# B&R Automation Studio project NAELD004C00R10L518F00 (part 48)

##### Act_OpsRun.st
```iecst
(** 2019-04-16 **)
ACTION Act_OpsRun:
	Act_LogStep;

	IF p_bOpsTravLifErrCmdUnclmp THEN //from travLif width chk error
		eMagConv2ClpAct :=	MagConv2ClpActStopClpr;

		IF (p_eMagConv2ClpStatus = Done AND p_eMagConv2ClpStat = MagConv2ClpActStopClpr) THEN

			eMagConv2ClpAct	:= MagConv2ClpActIdle;
			bPneuUnclmpDone := TRUE; //to travlif
		END_IF
	END_IF

	IF eGotoOpsStep <> eOpsStep THEN

		CASE eGotoOpsStep OF
			MagConvLDStepSelClampCtrl:
				IF p_bMagOrientChkSenPrep THEN
					//checking orientation of mag
					IF p_bMagHeightDetEn AND p_bMagHeightDetPrep THEN

						IF p_bMag3OrientationChkSen1 AND p_bMagHeightDetSen3 THEN // Magazine Type Check with height Detection Sensor
							eOpsStep := eGotoOpsStep;
						ELSE
							eMagConv2ClpAct :=	MagConv2ClpActStopClpr;

							IF (p_eMagConv2ClpStatus = Done AND p_eMagConv2ClpStat = MagConv2ClpActStopClpr) THEN

								eMagConv2ClpAct	:= MagConv2ClpActIdle;
								eStatus		:= Error;
								udiStatus	:= 10008;	//'Wrong Magazine Orientation Placed Or Wrong Magazine Loaded'
							END_IF
						END_IF

					ELSE

						IF p_bMag3OrientationChkSen1 AND NOT p_bMagHeightDetSen3 THEN //Without Check Height Detection Sensor
							eOpsStep := eGotoOpsStep;
						ELSE
							eMagConv2ClpAct :=	MagConv2ClpActStopClpr;
							eSelClampCtrl := PneuActExt; //unclmp
							IF (p_eMagConv2ClpStatus = Done AND p_eMagConv2ClpStat = MagConv2ClpActStopClpr) THEN

								eMagConv2ClpAct	:= MagConv2ClpActIdle;
								eStatus		:= Error;
								udiStatus	:= 10008;	//'Wrong Magazine Orientation Placed Or Wrong Magazine Loaded'
							END_IF
						END_IF

					END_IF
				ELSE
					eOpsStep	:= eGotoOpsStep;
				END_IF

			MagConvLDStepMagExitClampCtrl: //For Siemen
				IF p_eNtParamCustomerReq = Siemens AND (eOpsStep <> MagConvLDStepMagExtMESStdByChk )
					AND (p_tyLocalBufferStat.bBffrMty OR p_bDISOTAGVReady)
					AND NOT(iMagMESAcptCond < 0)AND p_bMcParamMesRFIDEn THEN
					eOpsStep := MagConvLDStepMagExtMESStdByChk;
					eGotoOpsStep := MagConvLDStepMagExtMESStdByChk; //exit mes
					//ePrevStepBeforeMESStdBy := MagConvLDStepMagExitClampCtrl;
				ELSE
					bExitDelAutoRcp := TRUE; 									//Clear the rcp and calc pitch
					eOpsStep	:= eGotoOpsStep;
				END_IF

			MagConvLDStepMagExitMnl:
				IF p_bRlsMag AND  p_eNtParamCustomerReq = Siemens AND eOpsStep <> MagConvLDStepMagExtMESStdByChk
					AND eOpsStep <> MagConvLDStepMagEntMESStdByChk AND p_bMcParamMesRFIDEn THEN
					eGotoOpsStep := MagConvLDStepMagExtMESStdByChk; //exit mes
				ELSE
					IF eOpsStep = MagConvLDStepMagExtMESStdByChk THEN
						ePrevStepBeforeMESStdBy := MagConvLDStepMagExitMnl;
					END_IF
					IF p_eNtParamCustomerReq = We_Fabricate  AND p_bMcParamMesRFIDEn THEN
						bExitDelAutoRcp := TRUE;
					END_IF
					eOpsStep	:= eGotoOpsStep;
				END_IF

			ELSE
				eOpsStep	:= eGotoOpsStep;

		END_CASE

	END_IF

	IF eOpsStep = eGotoOpsStep THEN

		IF bPaused = FALSE THEN

			CASE eOpsStep OF

				MagSetupULStepInitPneu:
					sStepTxt	:= 'Initializing Pneumatic';

					p_usiMagConv := 3;
					CASE p_usiMagConv OF
						1:
							p_tyLocalBufferStat ACCESS ADR(p_tyBufferStat1);
							p_bLocalMagEntrySen ACCESS ADR(p_bMagEntrySen1);
							p_bLocalBufferMagPresent ACCESS ADR(p_bBufferMagPresent1);
							p_dtLocalBufferMagPresentTm ACCESS ADR(p_dtBufferMagPresentTm1);
						2:
							p_tyLocalBufferStat ACCESS ADR(p_tyBufferStat2);
							p_bLocalMagEntrySen ACCESS ADR(p_bMagEntrySen2);
							p_bLocalBufferMagPresent ACCESS ADR(p_bBufferMagPresent2);
							p_dtLocalBufferMagPresentTm ACCESS ADR(p_dtBufferMagPresentTm2);
						3:
							p_tyLocalBufferStat ACCESS ADR(p_tyBufferStat3);
							p_bLocalMagEntrySen ACCESS ADR(p_bMagEntrySen3);
							p_bLocalBufferMagPresent ACCESS ADR(p_bBufferMagPresent3);
							p_dtLocalBufferMagPresentTm ACCESS ADR(p_dtBufferMagPresentTm3);
						4:
							p_tyLocalBufferStat ACCESS ADR(p_tyBufferStat4);
							p_bLocalMagEntrySen ACCESS ADR(p_bMagEntrySen4);
							p_bLocalBufferMagPresent ACCESS ADR(p_bBufferMagPresent4);
							p_dtLocalBufferMagPresentTm ACCESS ADR(p_dtBufferMagPresentTm4);
					END_CASE
					IF p_bProjLifTravMnlLoad = FALSE THEN
						eSafetyBarAct	:= PneuActExt;
					ELSE
						eGotoOpsStep := MagConvLDStepMagUSComm;
					END_IF
					IF (p_eSafetyBarStatus = Done AND p_eSafetyBarStat = PneuActExt) THEN
						eSafetyBarAct	:= PneuActIdle;
						eGotoOpsStep	:= MagConvLDStepInitMag;

						bPaused	:= p_bStop OR p_bStep;
					END_IF

				MagConvLDStepInitMag:
					sStepTxt	:= 'Initializing Magazine';
					IF p_bProjLifTravMnlLoad = TRUE THEN
						eGotoOpsStep := MagConvLDStepMagUSComm;
					ELSIF bMagExitedWait THEN
						eGotoOpsStep	:= MagConvLDStepMagExitedWait;
						//eGotoOpsStep	:= MagConvLDStepInitMagEnt;
					ELSIF (ePrevStepBeforeMESStdBy = MagConvLDStepMagExitMnl AND p_bLinkDIMagPresentSen3) OR (p_bHCommModChg AND p_bLinkDIMagPresentSen3)THEN
						eGotoOpsStep	:= MagConvLDStepMagExitMnl;
					ELSIF p_bNtParamAutoRcpPrep AND p_bHermesSvyPrep AND p_bMcParamHermesSvyEn THEN
						bHCommModChgDone := TRUE; //to UI
						eGotoOpsStep	:= MagConvLDStepInitMagConv;
					ELSE
						bHCommModChgDone := TRUE; //to UI
						eGotoOpsStep	:= MagConvLDStepInitSetMagFull;
					END_IF

					bPaused	:= p_bStop OR p_bStep;

				MagConvLDStepInitMagEnt:
					sStepTxt	:= 'Initializing Magazine Conveyor';
					eMagConv2ClpAct	:= MagConv2ClpActInit;
					IF (p_eMagConv2ClpStatus = Done AND p_eMagConv2ClpStat = MagConv2ClpActInit) THEN
						eMagConv2ClpAct	:= MagConv2ClpActIdle;
						IF p_bMagConv2ClpHvMag = FALSE THEN
							eGotoOpsStep	:= MagConvLDStepMagUSComm;
						ELSE
							eGotoOpsStep	:= MagConvLDStepInitMagFixClp;
						END_IF
					END_IF

				MagConvLDStepInitMagFixClp:
					sStepTxt	:= 'Initializing Fixed Clamp';
					eMagConv2ClpAct	:= MagConv2ClpActFixClprClamp;
					IF (p_eMagConv2ClpStatus = Done AND p_eMagConv2ClpStat = MagConv2ClpActFixClprClamp) THEN
						eMagConv2ClpAct	:= MagConv2ClpActIdle;
						IF bMagAutoEx THEN
							eDSSOTAct	:= SOTActRun;
						ELSE
							eDSSOTAct	:= SOTActIdle;
						END_IF

						IF p_bDIMagConvCAB717Sen THEN
							bMagSizeLarge := TRUE;
						ELSE
							bMagSizeLarge := FALSE;
						END_IF
						eGotoOpsStep	:= MagConvLDStepSelClampCtrl;
					END_IF

				MagConvLDStepInitSetMagFull	:
					sStepTxt	:= 'Set Magazine Full';
					IF bSetMagFull AND p_tyBufferStat3.diTtlBrdCap = 1 THEN
						eBufferAct := BufferActSetFull;
						IF p_eBufferStat = BufferActSetFull AND p_eBufferStatus = Done THEN
							bSetMagFull := FALSE;
							eBufferAct := BufferActIdle;
							eGotoOpsStep	:= MagConvLDStepInitMagConv;
						END_IF
					ELSIF bSetMagFull AND p_tyBufferStat3.diTtlBrdCap <> 1 THEN
						bSetMagFull := FALSE;
						eBufferAct := BufferActIdle;
						eGotoOpsStep	:= MagConvLDStepInitMagConv;
					ELSE
						bSetMagFull := FALSE;
						eBufferAct := BufferActIdle;
						eGotoOpsStep	:= MagConvLDStepInitMagConv;
					END_IF
					bPaused	:= p_bStop OR p_bStep;

				MagConvLDStepInitMagConv:
					sStepTxt	:= 'Initializing Magazine Conveyor';

					eMagConv2ClpAct	:= MagConv2ClpActInitStopClp;
					eSelClampCtrl := PneuActExt;

					IF (p_eMagConv2ClpStatus = Done AND p_eMagConv2ClpStat = MagConv2ClpActInitStopClp)
						AND (p_eSelClampCtrlStat = PneuActExt AND p_eSelClampCtrlStatus = Done)
						THEN
						eSelClampCtrl	:= PneuActIdle;
						eMagConv2ClpAct	:= MagConv2ClpActIdle;

						IF p_bMagConv2ClpHvMag = FALSE THEN
							eGotoOpsStep	:= MagConvLDStepMagUSComm;
							bExitDelAutoRcp := TRUE;
							usiAccWO := 0;
							ePrevStepBeforeMESStdBy := MagConvLDStepNA; //finish exit from extMes
						ELSE
						//	eGotoOpsStep		:= MagConvLDStepBffrStatChk;
							eGotoOpsStep		:= MagConvLDStepSelClampCtrl;
						END_IF

						bPaused	:= p_bStop OR p_bStep;

					END_IF

				MagConvLDStepSafetyBarExtCtrl:
					eSafetyBarAct	:= PneuActExt;

					IF(p_eSafetyBarStatus = Done AND p_eSafetyBarStat = PneuActExt)
						THEN
						eSafetyBarAct	:= PneuActIdle;
						eGotoOpsStep	:= MagConvLDStepMagUSComm;
					END_IF

				MagConvLDStepMagUSComm:
					sStepTxt	:= 'Communicating AIV And Ready Transport In Magazine';

					eAGVMagAct	:= AGVMagActEnter;
					IF bMagAutoEx THEN
						eUSSOTAct	:= SOTActRun;
					ELSE
						eUSSOTAct	:= SOTActIdle;
					END_IF
					eDSSOTAct	:= SOTActIdle;
					bMagSizeLarge := FALSE;
					bMagExitedWait	:= FALSE;

					IF p_bSafetyBarExtended = FALSE THEN
						eGotoOpsStep	:= MagConvLDStepSafetyBarExtCtrl;
					ELSIF p_bAGVMagMcRunRdy = TRUE OR p_bUSSOTTransporting= TRUE THEN
						eGotoOpsStep	:= MagConvLDStepMagEnt;

					ELSIF p_bNewMag = TRUE OR bNewMagAutoDetected = TRUE THEN
						eAGVMagAct		:= AGVMagActIdle;
						eGotoOpsStep	:= MagConvLDStepMagEntMnl;

					ELSE
						bPaused	:= p_bStop;

						IF bPaused = TRUE THEN
							eAGVMagAct	:= AGVMagActIdle;
							eUSSOTAct	:= SOTActIdle;
						END_IF

					END_IF

				MagConvLDStepMagEnt:

					IF p_bUSSOTConvStart THEN
						sStepTxt	:= 'Conveyor Entering Magazine To End';
						eMagConv2ClpAct	:= MagConv2ClpActEntStopClp;

					ELSIF bNewMagAutoDetected = TRUE THEN
						eAGVMagAct			:= AGVMagActIdle;
						eGotoOpsStep		:= MagConvLDStepMagEntMnl;

					ELSIF p_bUSSOTConvStop THEN
						sStepTxt	:= 'Conveyor Stopping';
						eMagConv2ClpAct	:= MagConv2ClpActStopClpr;
						IF (p_eMagConv2ClpStatus = Done AND p_eMagConv2ClpStat = MagConv2ClpActEntStopClp) THEN
							eMagConv2ClpAct		:= MagConv2ClpActIdle;

						END_IF
					END_IF

					IF (p_eMagConv2ClpStatus = Done AND p_eMagConv2ClpStat = MagConv2ClpActEntStopClp) THEN
						eAGVMagAct			:= AGVMagActIdle;
						eMagConv2ClpAct		:= MagConv2ClpActIdle;
						eUSSOTAct			:= SOTActIdle;
						eGotoOpsStep		:= MagConvLDStepSelClampCtrl;
						bPaused	:= p_bStop OR p_bStep;

					ELSE

					END_IF

				MagConvLDStepMagEntMnl:
					sStepTxt	:= 'Magazine Conveyor Entering Magazine Manually';
					IF p_bProjLifTravMnlLoad = FALSE THEN
						eMagConv2ClpAct	:= MagConv2ClpActEntStopClp;
					ELSE
						eGotoOpsStep		:= MagConvLDStepSelClampCtrl;
					END_IF
					IF p_eMagConv2ClpStatus = Done AND p_eMagConv2ClpStat = MagConv2ClpActEntStopClp THEN

						eMagConv2ClpAct		:= MagConv2ClpActIdle;
						eGotoOpsStep		:= MagConvLDStepSelClampCtrl;
						eUSSOTAct			:= SOTActIdle;
						eAGVMagAct			:= AGVMagActIdle;
						bPaused	:= p_bStop OR p_bStep;
					END_IF

				MagConvLDStepSelClampCtrl:
					sStepTxt	:= 'Magazine Selection Control';
					bNewMagVerifyStarted := TRUE;
					bExitDelAutoRcp := FALSE;

					CASE p_bLinkMagRcpCurrRcpMagModel OF
						0: //CAB706.2
							IF p_bDIMagConvCAB717Sen = FALSE THEN
								eSelClampCtrl := PneuActRet;
							END_IF
							eGotoOpsStep	:= MagConvLDStepVerifyMag;

						1: //CAB716.2
							IF p_bDIMagConvCAB717Sen = FALSE THEN
								eSelClampCtrl := PneuActRet;
							END_IF
							eGotoOpsStep	:= MagConvLDStepVerifyMag;

						2: //CAB717.2
							eSelClampCtrl 	:= PneuActExt;
							eGotoOpsStep	:= MagConvLDStepVerifyMag;

					END_CASE

					bPaused	:= p_bStop OR p_bStep;

				MagConvLDStepVerifyMag:
					sStepTxt	:= 'Magazine Model Verification';

					bNewMagVerifyStarted := TRUE;
					fbWrongMagTm(IN:= bNewMagVerified = FALSE);
					IF fbWrongMagTm.Q AND NOT bMagExitedWait  THEN
						fbWrongMagTm(IN:= FALSE);
						eGotoOpsStep		:= MagConvLDStepMagExitMnl;
					ELSIF bMagExitedWait OR ePrevStepBeforeMESStdBy = MagConvLDStepMagExitMnl THEN //added extMes true
						eGotoOpsStep		:= MagConvLDStepMagExitMnl;
					ELSIF bNewMagVerified AND NOT bMagExitedWait THEN
						fbSelClmpTm(IN:= TRUE);
						IF fbSelClmpTm.Q THEN
							fbSelClmpTm(IN:= FALSE);
							eSelClampCtrl	:= PneuActIdle;
							IF (p_eNtParamCustomerReq = Siemens AND p_bMcParamHermesSvyEn AND p_bHermesSvyPrep) OR
								(p_eNtParamCustomerReq = We_Fabricate AND p_bMcParamMesRFIDEn) THEN
								IF  (iMagMESAcptCond > 0 OR usiAccWO > 0 OR bWriteRFID) AND iMagMESAcptCond <> 255 THEN
									p_bAutoRcpbMag3RcpLoaded := FALSE; //bi-dir
									eGotoOpsStep		:= MagConvLDStepBffrStatChk;
								ELSIF iMagMESAcptCond = 0 OR usiAccWO = 0 THEN
									bQueryWO := TRUE;
									eGotoOpsStep		:= MagConvLDStepMagEntMESStdByChk;
								END_IF
							ELSE
								eGotoOpsStep		:= MagConvLDStepBffrStatChk;
							END_IF
						END_IF

					END_IF

					IF p_bDIMagConvCAB717Sen THEN
						bMagSizeLarge := TRUE;
					ELSE
						bMagSizeLarge := FALSE;
					END_IF

//					IF bNewMagVerified AND p_eSelClampCtrlStatus = Done THEN
//
//						eSelClampCtrl	:= PneuActIdle;
//						eGotoOpsStep	:= MagConvLDStepBffrStatChk;
//					END_IF
					bPaused	:= p_bStop OR p_bStep;

				MagConvLDStepMagEntMESStdByChk:
					sStepTxt	:= 'Read RFID and Query Work Order';
					bReadRFID := TRUE;
					fbReadRFIDTO(IN:= bReadRFID);
					iMagMESAcptCond := INT_TO_USINT(p_tyResponseFromMES.iAcceptCondition);
					IF (p_tyResponseFromMES.iAcceptCondition > 0 AND p_eNtParamCustomerReq = We_Fabricate) OR p_bAutoRcpbMag3RcpLoaded THEN //Accept or rcv sendWO
						usiAccWO := 1;
						bQueryWO := FALSE;
						p_bAutoRcpbMag3RcpLoaded := FALSE; //bi-dir
						eGotoOpsStep := MagConvLDStepAutoRcpSetMagFull;
					//	eGotoOpsStep := MagConvLDStepBffrStatChk;
					ELSIF p_tyResponseFromMES.iAcceptCondition < 0  THEN						//No Accept (-1)
						eAGVMagAct	:= AGVMagActExit;
						IF p_bRlsMag THEN
							p_bRlsMag := FALSE; //bi-dir
							bQueryWO := FALSE;
							eGotoOpsStep	:= MagConvLDStepMagExitMnl;
						ELSIF p_bAGVMagMcRunRdy = TRUE THEN
							bQueryWO := FALSE;
							eGotoOpsStep	:= MagConvLDStepMagMtyExit;
						END_IF
					ELSIF fbReadRFIDTO.Q THEN
						sStepTxt	:= 'Wait For Read RFID';
						IF p_bRlsMag THEN
							p_bRlsMag := FALSE; //bi-dir
							bQueryWO := FALSE;
							eGotoOpsStep	:= MagConvLDStepMagExitMnl;
						END_IF
					END_IF
					IF eGotoOpsStep <> MagConvLDStepMagEntMESStdByChk THEN
						bReadRFID := FALSE;
						fbReadRFIDTO(IN:= bReadRFID);//false
					END_IF
					IF p_eNtParamCustomerReq = We_Fabricate THEN
						sStepTxt	:= 'Wait For MES feedback';
					END_IF

					bPaused	:= p_bStop OR p_bStep;

				MagConvLDStepAutoRcpSetMagFull:
					sStepTxt	:= 'Set Magazine Full';
					eBufferAct := BufferActSetFull;
					IF p_eBufferStat = BufferActSetFull AND p_eBufferStatus = Done THEN
						eBufferAct := BufferActIdle;
						IF p_ausiSvyMagAccOrder[3] = 10 OR p_ausiLCSLFMagAccOrder[3] = 10 THEN //working number
							eGotoOpsStep := MagConvLDStepBffrStatChk;
						END_IF
					END_IF
					bPaused	:= p_bStop OR p_bStep;

				MagConvLDStepBffrStatChk:
					sStepTxt	:= 'Checking Buffer Status';

					IF p_eBufferStatus = Idle THEN

						IF (p_tyLocalBufferStat.bBffrMty = TRUE OR p_bUSAllow = FALSE) THEN
							//eGotoOpsStep	:= MagConvLDStepMagMtyDSComm;
							eGotoOpsStep	:= MagConvLDStepMagExitClampCtrl;
						ELSE
							eGotoOpsStep	:= MagConvLDStepSafetyBarRetCtrl;
						END_IF

						bPaused	:= p_bStop OR p_bStep;

					END_IF

				MagConvLDStepSafetyBarRetCtrl:
					eSafetyBarAct	:= PneuActRet;

					IF (p_eSafetyBarStatus = Done AND p_eSafetyBarStat = PneuActRet) THEN
						eSafetyBarAct	:= PneuActIdle;
						eGotoOpsStep	:= MagConvLDStepPreNxtUnlBffr;

						bPaused	:= p_bStop OR p_bStep;
					END_IF

				MagConvLDStepPreNxtUnlBffr:
					sStepTxt	:= 'Computing Next Unload Buffer';

					eBufferAct	:= BufferActNxtUnload;

					IF p_eBufferStatus = Done AND p_eBufferStat = BufferActNxtUnload THEN
						eBufferAct		:= BufferActIdle;
						eGotoOpsStep	:= MagConvLDStepMagCmp;

						bPaused	:= p_bStop OR p_bStep;
					END_IF

				MagConvLDStepMagCmp:
					sStepTxt	:= 'Comparing Magazine';

					a_tyMagAllwBffrStat[1]	:= p_tyBufferStat1;
					a_tyMagAllwBffrStat[2]	:= p_tyBufferStat2;
					a_tyMagAllwBffrStat[3]	:= p_tyBufferStat3;
					a_tyMagAllwBffrStat[4]	:= p_tyBufferStat4;

					a_bMagAllwMagClamped[1]	:= p_bMagClampRS1;
					a_bMagAllwMagClamped[2]	:= p_bMagClampRS2;
					a_bMagAllwMagClamped[3]	:= p_bMagClampRS3;
					a_bMagAllwMagClamped[4]	:= p_bMagClampRS4;

					a_bMagAllwMagPresent[1]	:= p_bBufferMagPresent1 AND NOT p_bLD1ExitedWait;
					a_bMagAllwMagPresent[2]	:= p_bBufferMagPresent2 AND NOT p_bLD2ExitedWait;
					a_bMagAllwMagPresent[3]	:= p_bBufferMagPresent3 AND NOT bMagExitedWait;
					a_bMagAllwMagPresent[4]	:= p_bBufferMagPresent4 AND NOT p_bLD4ExitedWait;

					a_udiMagAllwMagPresentTm[1]	:= DT_TO_UDINT(p_dtBufferMagPresentTm1);
					a_udiMagAllwMagPresentTm[2]	:= DT_TO_UDINT(p_dtBufferMagPresentTm2);
					a_udiMagAllwMagPresentTm[3]	:= DT_TO_UDINT(p_dtBufferMagPresentTm3);
					a_udiMagAllwMagPresentTm[4]	:= DT_TO_UDINT(p_dtBufferMagPresentTm4);
					//Sorting Priority
					memset(ADR(a_udiMagAllwPriority), 0, SIZEOF(a_udiMagAllwPriority));

					IF (p_bMcParamHermesSvyEn AND p_bNtParamAutoRcpPrep) OR (p_bMcParamMesRFIDEn AND p_eNtParamCustomerReq = We_Fabricate) THEN
						FOR udi :=1 TO 3 DO
							IF p_ausiSvyMagAccOrder[udi] = 10 OR p_ausiLCSLFMagAccOrder[udi] = 10 THEN
								a_udiMagAllwPriority[udi] :=  1;
							ELSE
								a_udiMagAllwPriority[udi] := 3;
							END_IF
						END_FOR

					ELSE // standard
						FOR udi := 1 TO 4 DO
							udiCount	:= 4;
							udiCmpTm	:= a_udiMagAllwMagPresentTm[udi];

							FOR udi1 := 1 TO 4 DO
								IF a_udiMagAllwMagPresentTm[udi1] > udiCmpTm THEN
									udiCount	:= udiCount - 1;
								END_IF
							END_FOR

							a_udiMagAllwPriority[udi]	:= udiCount;
						END_FOR
						FOR udi := 4 TO 1 BY -1 DO
							FOR udi1 := 4 TO 1 BY -1 DO
								IF (udi <> udi1) AND (a_udiMagAllwPriority[udi] = a_udiMagAllwPriority[udi1]) THEN
									a_udiMagAllwPriority[udi1]	:= a_udiMagAllwPriority[udi1] - 1;
								END_IF
							END_FOR
						END_FOR
					END_IF

					//Checking Buffer Status
					memset(ADR(a_udiMagAllwSum), 0, SIZEOF(a_udiMagAllwSum));

					FOR udi := 1 TO 4 DO
						//Priority
						a_udiMagAllwSum[udi]	:= a_udiMagAllwSum[udi] + a_udiMagAllwPriority[udi];
						//Enable
						IF pa_bMagDis[udi] = FALSE THEN
							a_udiMagAllwSum[udi]	:= a_udiMagAllwSum[udi] + 1000;
						END_IF
						//Magazine Clamped
						IF a_bMagAllwMagClamped[udi] = TRUE THEN
							a_udiMagAllwSum[udi]	:= a_udiMagAllwSum[udi] + 1000;
						END_IF
						//Magazine Present
						IF a_bMagAllwMagPresent[udi] = TRUE THEN
							a_udiMagAllwSum[udi]	:= a_udiMagAllwSum[udi] + 1000;
						END_IF
						//Magazine Full
						IF a_tyMagAllwBffrStat[udi].bBffrFull = TRUE THEN
							a_udiMagAllwSum[udi]	:= a_udiMagAllwSum[udi] + 2500;
						END_IF
						//Magazine Available
						IF a_tyMagAllwBffrStat[udi].bBffrFull = FALSE AND a_tyMagAllwBffrStat[udi].bBffrMty = FALSE THEN
							a_udiMagAllwSum[udi]	:= a_udiMagAllwSum[udi] + 3000;
						END_IF
					END_FOR

					udiMagAllwGo	:= 99;

					FOR udi := 1 TO 4 DO
						//Enable + Magazine Clamped + Magazine Present + Magazine Available
						IF a_udiMagAllwSum[udi] >= 6000 THEN

							IF udiMagAllwGo <> 99 THEN
								//Priority
								IF a_udiMagAllwSum[udi] < a_udiMagAllwSum[udiMagAllwGo] THEN
									udiMagAllwGo	:= udi;
								END_IF
							ELSE
								udiMagAllwGo	:= udi;
							END_IF

						END_IF

					END_FOR

					IF udiMagAllwGo = 99 THEN

						FOR udi := 1 TO 4 DO
							//Enable + Magazine Clamped + Magazine Present + Magazine Full
							IF a_udiMagAllwSum[udi] >= 5500 THEN

								IF udiMagAllwGo <> 99 THEN
									//Priority
									IF a_udiMagAllwSum[udi] < a_udiMagAllwSum[udiMagAllwGo] THEN
										udiMagAllwGo	:= udi;
									END_IF
								ELSE
									udiMagAllwGo	:= udi;
								END_IF

							END_IF

						END_FOR

					END_IF

					IF p_bRlsMag = TRUE THEN
						eGotoOpsStep	:= MagConvLDStepMagExitMnl;

					ELSIF p_bDISOTAGVReady AND p_eNtParamCustomerReq = Siemens THEN
						eGotoOpsStep	:= MagConvLDStepMagExitClampCtrl;

					ELSIF (p_tyLocalBufferStat.bBffrMty = TRUE OR p_bUSAllow = FALSE) AND p_bInShutterExtended THEN
					//	eGotoOpsStep    := MagConvLDStepMagMtyDSComm;
						eGotoOpsStep    := MagConvLDStepMagExitClampCtrl;
					ELSE

						IF udiMagAllwGo <> 99 THEN

							IF udiMagAllwGo = p_usiMagConv (*AND p_eOpsTravLifLDPosGo = TravLifLDPosUS3*) THEN
								bMagBffrAvl		:= TRUE;
								eGotoOpsStep	:= MagConvLDStepNxtUnloadBffr;

								bPaused	:= p_bStop OR p_bStep;
							ELSE
								bPaused	:= p_bStop;
							END_IF

						ELSE
							bPaused	:= p_bStop;
						END_IF

					END_IF

				MagConvLDStepNxtUnloadBffr:
					sStepTxt	:= 'Computing Next Unload Buffer';

					eBufferAct	:= BufferActNxtUnload;

					IF p_eBufferStatus = Done AND p_eBufferStat = BufferActNxtUnload THEN
						eBufferAct		:= BufferActIdle;
						eGotoOpsStep	:= MagConvLDStepBffrDSComm;

						bPaused	:= p_bStop OR p_bStep;
					END_IF

				MagConvLDStepBffrDSComm:
					sStepTxt	:= 'Communicating Buffer Downstream';

//					IF (p_tyBufferStat2.bBffrFull OR p_bBufferMagPresent2 = FALSE)
//						AND (p_tyBufferStat3.bBffrFull OR p_bBufferMagPresent3 = FALSE)
//						THEN
//						eDSSMEMAAct	:= SMEMAActRun;
//					END_IF

					eDSSMEMAAct	:= SMEMAActRun;

					IF p_bDSSMEMAConvStart = TRUE THEN
						eGotoOpsStep	:= MagConvLDStepBffrExitBrd;

					ELSIF bOpsTravLifULUpdatePullSlot AND p_eOpsTravLifLDPosGo = TravLifLDPosUS3 THEN
						bMagBffrAvl		:= FALSE;
						IF p_tyLocalBufferStat.bBffrMty = FALSE AND p_bUIP800Press3 = FALSE THEN
							eGotoOpsStep	:= MagConvLDStepUnloadBffr;
						ELSE
							eGotoOpsStep	:= MagConvLDStepBffrStatChk;
							bMagBffrAvl		:= FALSE;
						END_IF

					ELSIF p_bRlsMag = TRUE THEN
						bMagBffrAvl		:= FALSE;
						eDSSMEMAAct		:= SMEMAActIdle;
						eGotoOpsStep	:= MagConvLDStepMagExitMnl;

					ELSIF (p_tyLocalBufferStat.bBffrMty = TRUE OR p_bUSAllow = FALSE) AND p_bInShutterExtended THEN
						bMagBffrAvl		:= FALSE;
						eDSSMEMAAct		:= SMEMAActIdle;
					//	eGotoOpsStep    := MagConvLDStepMagMtyDSComm;
						eGotoOpsStep    := MagConvLDStepMagExitClampCtrl;
					ELSE

						IF pa_bMagDis[usiMagConv] = TRUE THEN		//Checking Magazine Enable
							bMagBffrAvl		:= FALSE;
				//			eGotoOpsStep	:= MagConvLDStepMagCmp;
							eGotoOpsStep	:= MagConvLDStepPreNxtUnlBffr;

							bPaused	:= p_bStop OR p_bStep;
						ELSE
							bPaused	:= p_bStop;
						END_IF

						IF bPaused = TRUE OR pa_bMagDis[usiMagConv] = TRUE THEN
							eDSSMEMAAct	:= SMEMAActIdle;
						END_IF

					END_IF

				MagConvLDStepBffrExitBrd:
					IF p_bDSSMEMAConvStart = TRUE THEN
						sStepTxt	:= 'Transferring Board Out From Magazine';
						IF p_bRlsMag = TRUE THEN
							bMagBffrAvl		:= FALSE;
							eDSSMEMAAct		:= SMEMAActIdle;
							eGotoOpsStep	:= MagConvLDStepMagExitMnl;
						END_IF
					END_IF

					IF p_eDSSMEMAStatus = Done AND p_eDSSMEMAStat = SMEMAActRun THEN
						eDSSMEMAAct		:= SMEMAActIdle;
						//	eGotoOpsStep	:= MagConvLDStepUnloadBffr;
						IF p_tyLocalBufferStat.bBffrMty = FALSE THEN
							eGotoOpsStep	:= MagConvLDStepUnloadBffr;
						ELSE
							eGotoOpsStep	:= MagConvLDStepBffrStatChk;
							bMagBffrAvl		:= FALSE;
						END_IF
					END_IF

				MagConvLDStepUnloadBffr:
					sStepTxt	:= 'Unloading Buffer';

						eBufferAct	:= BufferActUnload;
						bOpsTravLifULUpdatePullSlot := FALSE;
						bMagBffrAvl		:= FALSE;
					IF p_eBufferStatus = Done AND p_eBufferStat = BufferActUnload THEN
						eBufferAct		:= BufferActIdle;
						bMagBffrAvl		:= FALSE;

							eGotoOpsStep	:= MagConvLDStepBffrStatChk;

						bPaused	:= p_bStop OR p_bStep;
					END_IF

				MagConvLDStepMagExtMESStdByChk:
					sStepTxt	:= 'Mag StdBy for MES response Before Exiting';
					bWriteRFID := TRUE;
					fbWriteRFIDTO(IN:= bWriteRFID ,PT:= DINT_TO_TIME(p_diRFIDTO));
					bExitDelAutoRcp := TRUE; 									//Clear the rcp and calc pitch
					IF p_tyResponseFromMES.bRFIDWriteComplete  THEN 			//Accept
//						IF ePrevStepBeforeMESStdBy = MagConvULStepMagExitMnl THEN
							eGotoOpsStep := MagConvLDStepMagExitMnl;//MagConvLDStepMagExitClampCtrl;
//						ELSIF ePrevStepBeforeMESStdBy = MagConvULStepMagExitClampCtrl THEN
//							eGotoOpsStep := MagConvLDStepMagExitClampCtrl;
//						END_IF
					ELSIF fbWriteRFIDTO.Q  THEN
						sStepTxt	:= 'MES response to Write RFID Timeout, Press Rls Mag to Manual Exit ';
						IF p_bEjectMag THEN
							eGotoOpsStep := MagConvLDStepMagExitMnl;
						END_IF
					END_IF
					IF eGotoOpsStep <> MagConvLDStepMagExtMESStdByChk THEN
						bWriteRFID := FALSE;
						fbWriteRFIDTO(IN:= bWriteRFID);

					END_IF
					bPaused	:= p_bStop OR p_bStep;

				MagConvLDStepMagExitClampCtrl:
					sStepTxt	:= 'Extending Selection Clamp';
					eSelClampCtrl := PneuActExt;
					eSafetyBarAct	:= PneuActExt;

					IF (p_eSelClampCtrlStat = PneuActExt AND p_eSelClampCtrlStatus = Done)
						AND(p_eSafetyBarStatus = Done AND p_eSafetyBarStat = PneuActExt)
						THEN
							eSelClampCtrl	:= PneuActIdle;
							eSafetyBarAct	:= PneuActIdle;
							eGotoOpsStep    := MagConvLDStepMagMtyDSComm;
							bPaused	:= p_bStop OR p_bStep;
					END_IF

				MagConvLDStepMagMtyDSComm:
					sStepTxt	:= 'Communicating AGV Machine And Ready Exit';

					eAGVMagAct	:= AGVMagActExit;
					IF bMagAutoEx THEN
						eDSSOTAct	:= SOTActRun;
					ELSE
						eDSSOTAct	:= SOTActIdle;
					END_IF

					IF p_bAGVMagMcRunRdy = TRUE THEN
						eGotoOpsStep	:= MagConvLDStepMagMtyExit;

					ELSIF p_bRlsMag = TRUE OR ((p_tyLocalBufferStat.bBffrMty OR p_bUSAllow = FALSE) AND p_bInShutterExtended) THEN
						eAGVMagAct		:= AGVMagActIdle;
						eGotoOpsStep	:= MagConvLDStepMagExitMnl;

					ELSE
						bPaused	:= p_bStop;

						IF bPaused = TRUE THEN
							eAGVMagAct	:= AGVMagActIdle;
							eDSSOTAct	:= SOTActIdle;
						END_IF

					END_IF

				MagConvLDStepMagMtyExit:
					sStepTxt	:= 'Magazine Conveyor Exiting Magazine';

					eMagConv2ClpAct	:= MagConv2ClpActExitClpr;
					eSelClampCtrl	:= PneuActExt;

					IF ((p_eAGVMagStatus = Done AND p_eAGVMagStat = AGVMagActExit)
						OR (p_eDSSOTStatus = Done AND p_eDSSOTStat = SOTActRun))
						AND (p_eMagConv2ClpStatus = Done AND p_eMagConv2ClpStat = MagConv2ClpActExitClpr)
						AND (p_eSelClampCtrlStatus = Done AND p_eSelClampCtrlStat = PneuActExt)
						THEN

						eDSSOTAct	:= SOTActIdle;
						eAGVMagAct		:= AGVMagActIdle;
						eMagConv2ClpAct	:= MagConv2ClpActIdle;
						eSelClampCtrl	:= PneuActIdle;
						eGotoOpsStep	:= MagConvLDStepMagExitedAGVWait;
						bMagSizeLarge	:= FALSE;

						bPaused	:= p_bStop OR p_bStep;
					END_IF

				MagConvLDStepMagExitedAGVWait:
					sStepTxt	:= 'Magazine Exited and Wait for AGV Leave';

					IF bAIVInPos = FALSE OR p_bBufferMagRemoved THEN
						usiAccWO := 0;
						bExitDelAutoRcp := FALSE;
						eGotoOpsStep	:= MagConvLDStepMagUSComm;
						eDSSOTAct	:= SOTActIdle;
					END_IF

					bPaused	:= p_bStop OR p_bStep;

				MagConvLDStepMagExitMnl:
					sStepTxt	:= 'Magazine Conveyor Exiting Magazine Manually';
					IF p_bProjLifTravMnlLoad = FALSE THEN
						eMagConv2ClpAct	:= MagConv2ClpActPreExitClpr;
						eSelClampCtrl	:= PneuActExt;
						eSafetyBarAct	:= PneuActExt;
					ELSE
						eGotoOpsStep    := MagConvLDStepMagExitedWait;
					END_IF
					IF ((p_eMagConv2ClpStatus = Done OR EDGENEG(p_bFixedSideDetect)) AND p_eMagConv2ClpStat = MagConv2ClpActPreExitClpr)
						AND (p_eSelClampCtrlStatus = Done AND p_eSelClampCtrlStat = PneuActExt)
						AND (p_eSafetyBarStatus = Done AND p_eSafetyBarStat = PneuActExt)
						THEN
						eSelClampCtrl	:= PneuActIdle;
						eSafetyBarAct	:= PneuActIdle;
						eMagConv2ClpAct	:= MagConv2ClpActIdle;

						eGotoOpsStep	:= MagConvLDStepMagExitedWait;

						bPaused	:= p_bStop OR p_bStep;
					END_IF

				MagConvLDStepMagExitedWait:
					sStepTxt	:= 'Magazine Exited And Waiting For Remove';
					eAGVMagAct	:= AGVMagActExit;
					IF bMagAutoEx THEN
						eDSSOTAct	:= SOTActRun;
					ELSE
						eDSSOTAct	:= SOTActIdle;
					END_IF
					bMagExitedWait	:= TRUE;
					bHCommModChgDone := TRUE; //to UI
					fbEntSenOff(IN:= p_bLocalMagEntrySen = FALSE);
					ePrevStepBeforeMESStdBy := MagConvLDStepNA; //finish exit from extMes
					iMagMESAcptCond := 0 ; //reset if 255 (-1)

					IF fbMagRemovedTm.Q OR fbEntSenOff.Q THEN
						usiAccWO := 0;
						bExitDelAutoRcp := FALSE;
						bMagExitedWait	:= FALSE;
						eGotoOpsStep	:= MagConvLDStepMagUSComm;
						eDSSOTAct	:= SOTActIdle;

					ELSIF p_bNewMag = TRUE THEN
						bMagExitedWait	:= FALSE;
						eAGVMagAct	:= AGVMagActIdle;
						eGotoOpsStep	:= MagConvLDStepMagEntMnl;
						eDSSOTAct	:= SOTActIdle;
					END_IF

					IF p_bAGVMagMcRunRdy = TRUE THEN
						eGotoOpsStep	:= MagConvLDStepMagMtyExit;
					ELSIF p_bDSSOTConvStart = TRUE THEN
						eGotoOpsStep	:= MagConvLDStepMagMtyExit;
					END_IF

					bPaused	:= p_bStop OR p_bStep;

			END_CASE

		END_IF

	END_IF

	bNewMagAllw	:= eOpsStep = MagConvLDStepMagUSComm;
	bRlsMagAllw	:= (eOpsStep = MagConvLDStepMagCmp
					OR eOpsStep = MagConvLDStepBffrDSComm
					OR eOpsStep = MagConvLDStepMagMtyDSComm
					OR eOpsStep = MagConvLDStepBffrExitBrd
					OR eOpsStep = MagConvLDStepMagEntMESStdByChk AND (p_tyResponseFromMES.iAcceptCondition < 0 OR fbReadRFIDTO.Q))
					AND NOT(p_bOpsTravLifLDEntBrd OR p_bOpsTravLifLDUSMagWidthChk OR p_bOpsTravLifMove)
					AND (p_bDIInShutterClosedRS OR p_bLinkProjCurtainSenPrep);

	Act_OpsInfo;

	//Operation State
	bOpsInitDone		:= eOpsStep > MagConvLDStepInitMagConv;
	bStepMagExitedWait	:= eOpsStep = MagConvLDStepMagExitedWait;
	bStepMagVerification:= eOpsStep = MagConvLDStepVerifyMag;
	bStepMagMtyExit		:= eOpsStep = MagConvLDStepMagMtyExit;
	bStepMagUSCom 		:= eOpsStep = MagConvLDStepMagUSComm;
	bStepDSCom 			:= eOpsStep = MagConvLDStepBffrDSComm;
	bAGVCommRdy			:= (eOpsStep = MagConvLDStepMagUSComm OR eOpsStep = MagConvLDStepMagMtyDSComm OR eOpsStep = MagConvLDStepMagExitedWait
							OR eOpsStep = MagConvLDStepMagEnt OR eOpsStep = MagConvLDStepMagMtyExit) AND p_bAGVMagMcRunRdy;
	bRlsMagBtnUnmask	:= eOpsStep = MagConvLDStepMagEntMESStdByChk AND (p_tyResponseFromMES.iAcceptCondition < 0 OR fbReadRFIDTO.Q) OR fbWriteRFIDTO.Q;
	bExtMesStdByChk		:= eOpsStep = MagConvLDStepMagExtMESStdByChk;
//	bExitDelAutoRcp	:= eOpsStep = MagConvLDStepMagMtyExit OR eOpsStep =  MagConvLDStepMagExitedWait OR eOpsStep =  MagConvLDStepMagExitedAGVWait
//							 OR eOpsStep = MagConvLDStepMagExitMnl;

END_ACTION
```

### OpsMagConvLD4.var - Change By Project
```iecst
(*2019-03-25*)
(**)
(*Action & State & Status*)
(**)
(*Alarm*)
VAR
	p_OpsMagConvLD4AlmData : UDINT;
	p_OpsMagConvLD4AlmData1 : UDINT;
END_VAR
(**)
(*Output*)
VAR
	p_OpsMagConvLD4StepTxt : UDINT;
	p_OpsMagConvLD4Paused : UDINT;
END_VAR
(**)
VAR
	p_OpsMagConvLD4BufferAct : UDINT;
	p_OpsMagConvLD4MagConv2ClpAct : UDINT;
	p_OpsMagConvLD4DSSMEMAAct : UDINT;
	p_OpsMagConvLD4AGVMagAct : UDINT;
	p_OpsMagConvLD4SafetyBarAct : UDINT;
END_VAR
(**)
VAR
	p_OpsMagConvLD4NewMagVerified : UDINT;
	p_OpsMagConvLD4MagMtyExit : UDINT;
	p_OpsMagConvLD4IncorrectMagModel : UDINT;
	p_OpsMagConvLD4MagSizeL : UDINT;
END_VAR
(**)
VAR
	p_OpsMagConvLD4InitDone : UDINT;
	p_OpsMagConvLD4MagBffrAvl : UDINT;
	p_OpsMagConvLD4NewMagAllw : UDINT;
	p_OpsMagConvLD4RlsMagAllw : UDINT;
	p_OpsMagConvLD4StepMagExitedWait : UDINT;
	p_OpsMagConvLD4StepUSCom : UDINT;
	p_OpsMagConvLD4StepSelClampCtrl : UDINT;
END_VAR
(**)
VAR
	p_OpsMagConvLD4USSOTAct : UDINT;
	p_OpsMagConvLD4DSSOTAct : UDINT;
	p_OpsMagConvLD4ExitedWait : UDINT;
	p_OpsMagConvLD4DSCom : UDINT;
END_VAR
```

### Program Logical/Operations/OpsMagConvLD4 (IEC) - 1.00.0 - 

#### InputRef.var
```iecst
(*2019-04-16*)
(**)
(*General*)
VAR
	p_udiRstErr : REFERENCE TO UDINT;
	p_bEn : REFERENCE TO BOOL;
	p_bDis : REFERENCE TO BOOL;
	p_bRun : REFERENCE TO BOOL;
	p_bStop : REFERENCE TO BOOL;
	p_bStep : REFERENCE TO BOOL;
END_VAR
(**)
(*Configuration*)
VAR
	p_sProgNm : REFERENCE TO STRING[15];
	p_bNtSettingsLoadDone : REFERENCE TO BOOL;
END_VAR
(**)
VAR
	p_usiMagConv : REFERENCE TO USINT;
	p_bInfoEn : REFERENCE TO BOOL;
	p_bInfoMag1Mty : REFERENCE TO BOOL;
	p_bInfoMag2Mty : REFERENCE TO BOOL;
	p_bInfoMag3Mty : REFERENCE TO BOOL;
END_VAR
(**)
VAR
	pa_bMagDis : REFERENCE TO ARRAY[1..4] OF BOOL;
END_VAR
(**)
VAR
	p_bNewMag : REFERENCE TO BOOL;
	p_bRlsMag : REFERENCE TO BOOL;
END_VAR
(**)
VAR
	p_tyBufferStat1 : REFERENCE TO tyBffrStat;
	p_tyBufferStat2 : REFERENCE TO tyBffrStat;
	p_tyBufferStat3 : REFERENCE TO tyBffrStat;
	p_tyBufferStat4 : REFERENCE TO tyBffrStat;
END_VAR
(**)
VAR
	p_bMagClampRS1 : REFERENCE TO BOOL;
	p_bMagClampRS2 : REFERENCE TO BOOL;
	p_bMagClampRS3 : REFERENCE TO BOOL;
	p_bMagClampRS4 : REFERENCE TO BOOL;
END_VAR
(**)
VAR
	p_bMagEntrySen1 : REFERENCE TO BOOL;
	p_bMagEntrySen2 : REFERENCE TO BOOL;
	p_bMagEntrySen3 : REFERENCE TO BOOL;
	p_bMagEntrySen4 : REFERENCE TO BOOL;
END_VAR
(**)
VAR
	p_bMagPresentSen1 : REFERENCE TO BOOL;
	p_bMagPresentSen2 : REFERENCE TO BOOL;
	p_bMagPresentSen3 : REFERENCE TO BOOL;
	p_bMagPresentSen4 : REFERENCE TO BOOL;
END_VAR
(**)
VAR
	p_bMagPresentSen : REFERENCE TO BOOL;
	p_bBufferMagPresent1 : REFERENCE TO BOOL;
	p_bBufferMagPresent2 : REFERENCE TO BOOL;
	p_bBufferMagPresent3 : REFERENCE TO BOOL;
	p_bBufferMagPresent4 : REFERENCE TO BOOL;
END_VAR
(**)
VAR
	p_dtBufferMagPresentTm1 : REFERENCE TO DATE_AND_TIME;
	p_dtBufferMagPresentTm2 : REFERENCE TO DATE_AND_TIME;
	p_dtBufferMagPresentTm3 : REFERENCE TO DATE_AND_TIME;
	p_dtBufferMagPresentTm4 : REFERENCE TO DATE_AND_TIME;
END_VAR
(**)
VAR
	p_eBufferStat : REFERENCE TO eBufferAction;
	p_eBufferStatus : REFERENCE TO eFBStatus;
END_VAR
(**)
VAR
	p_bBufferMagRemoved : REFERENCE TO BOOL;
END_VAR
(**)
VAR
	p_eMagConv2ClpStat : REFERENCE TO eMagConv2ClpAction;
	p_eMagConv2ClpStatus : REFERENCE TO eFBStatus;
	p_bMagConv2ClpHvMag : REFERENCE TO BOOL;
END_VAR
(**)
VAR
	p_eDSSMEMAStat : REFERENCE TO eSMEMAAction;
	p_eDSSMEMAStatus : REFERENCE TO eFBStatus;
	p_bDSSMEMAConvStart : REFERENCE TO BOOL;
END_VAR
(**)
VAR
	p_eAGVMagStat : REFERENCE TO eAGVMagAction;
	p_eAGVMagStatus : REFERENCE TO eFBStatus;
	p_bAGVMagMcRunRdy : REFERENCE TO BOOL;
	p_tyAGVToDTMag : REFERENCE TO tyTagAGVToDTMag;
END_VAR
(**)
VAR
	p_eSelClampCtrlStat : REFERENCE TO ePneuAction;
	p_eSelClampCtrlStatus : REFERENCE TO eFBStatus;
END_VAR
(**)
VAR
	p_bDIMagConvHeightSen : REFERENCE TO BOOL;
	p_bDIMagConvSelUnclampRS : REFERENCE TO BOOL;
	p_bDIMagConvCAB717Sen : REFERENCE TO BOOL;
	p_bDIMagConvSmallSen : REFERENCE TO BOOL;
	p_bDIMagConvLargeSen : REFERENCE TO BOOL;
	p_bDIInShutterClosedRS : REFERENCE TO BOOL;
END_VAR
(**)
VAR
	p_bOpsTravLifLDInitDone : REFERENCE TO BOOL;
END_VAR
(**)
VAR
	p_eUSSOTStat : REFERENCE TO eSOTAction;
	p_eUSSOTStatus : REFERENCE TO eFBStatus;
	p_bUSSOTTransporting : REFERENCE TO BOOL;
	p_bUSSOTConvStart : REFERENCE TO BOOL;
	p_bUSSOTConvStop : REFERENCE TO BOOL;
	p_bUSSOTUSRdy : REFERENCE TO BOOL;
	p_bUSSOTUSLargeMagRdy : REFERENCE TO BOOL;
END_VAR
(**)
VAR
	p_eDSSOTStat : REFERENCE TO eSOTAction;
	p_eDSSOTStatus : REFERENCE TO eFBStatus;
	p_bDSSOTConvStart : REFERENCE TO BOOL;
	p_bDSSOTConvStop : REFERENCE TO BOOL;
END_VAR
(**)
VAR
	p_bDISOTRcv : REFERENCE TO BOOL;
	p_bInShutterExtended : REFERENCE TO BOOL;
	p_bUSAllow : REFERENCE TO BOOL;
END_VAR
(**)
VAR
	p_bLD1ExitedWait : REFERENCE TO BOOL;
	p_bLD2ExitedWait : REFERENCE TO BOOL;
	p_bLD3ExitedWait : REFERENCE TO BOOL;
END_VAR
(**)
VAR
	p_eSafetyBarStat : REFERENCE TO ePneuAction;
	p_eSafetyBarStatus : REFERENCE TO eFBStatus;
	p_bSafetyBarExtended : REFERENCE TO BOOL;
	p_bSafetyBarRetracted : REFERENCE TO BOOL;
	p_bOpsTravLifULUpdatePullSlot : REFERENCE TO BOOL;
	p_bProjLifTravMnlLoad : REFERENCE TO BOOL;
END_VAR
(**)
(**)
```

#### InputRef_Link.var
```iecst
(*2020-05-20*)
(**)
(*External Data*)
VAR
	p_bLinkDIMagPresentSen1 : REFERENCE TO BOOL;
	p_bLinkMagConv2Clp1MtrIn : REFERENCE TO BOOL;
	p_bLinkMagConv2Clp1MtrOut : REFERENCE TO BOOL;
	p_bLinkDIMagPresentSen2 : REFERENCE TO BOOL;
	p_bLinkMagConv2Clp2MtrIn : REFERENCE TO BOOL;
	p_bLinkMagConv2Clp2MtrOut : REFERENCE TO BOOL;
	p_bLinkDIMagPresentSen3 : REFERENCE TO BOOL;
	p_bLinkMagConv2Clp3MtrIn : REFERENCE TO BOOL;
	p_bLinkMagConv2Clp3MtrOut : REFERENCE TO BOOL;
	p_bLinkDIMagPresentSen4 : REFERENCE TO BOOL;
	p_bLinkMagConv2Clp4MtrIn : REFERENCE TO BOOL;
	p_bLinkMagConv2Clp4MtrOut : REFERENCE TO BOOL;
	p_bLinkFixedMagClampRS1 : REFERENCE TO BOOL;
	p_bLinkRmtMagClampRS1 : REFERENCE TO BOOL;
	p_bLinkFixedMagClampRS2 : REFERENCE TO BOOL;
	p_bLinkRmtMagClampRS2 : REFERENCE TO BOOL;
	p_bLinkFixedMagClampRS3 : REFERENCE TO BOOL;
	p_bLinkRmtMagClampRS3 : REFERENCE TO BOOL;
	p_bLinkFixedMagClampRS4 : REFERENCE TO BOOL;
	p_bLinkRmtMagClampRS4 : REFERENCE TO BOOL;
	p_bLinkMcParamMagAutoDetTm : REFERENCE TO DINT;
	p_bLinkDIMagEntrySen : REFERENCE TO BOOL;
	p_bLinkNtParamMagModelAutoVerify : REFERENCE TO BOOL;
	p_bLinkMagRcpCurrRcpMagModel : REFERENCE TO USINT;
	p_bLinkNewMagVerified1 : REFERENCE TO BOOL;
	p_bLinkNewMagVerified2 : REFERENCE TO BOOL;
	p_bLinkNewMagVerified3 : REFERENCE TO BOOL;
END_VAR
(**)
VAR
	p_eLinkMag : REFERENCE TO eLDMag;
	p_usiLinkMod : REFERENCE TO USINT;
	p_bLinkMagRcpCurrRcpMagModel1 : REFERENCE TO USINT;
	p_eLinkMcParamMagExMode : REFERENCE TO eMcMagExchangeMode;
END_VAR
```

#### Local.var
```iecst
(*2019-04-16*)
(**)
(*Local Action, State & Status*)
VAR
	eStatus : eFBStatus := Idle;
	udiStatus : UDINT := 0;
	udiStatus1 : UDINT := 0;
END_VAR
(**)
(*Local Alarm*)
VAR
	tyAlmData : tyAlmDat;
	tyAlmData1 : tyAlmDat;
	a_tyAlmText : ARRAY[10000..10099] OF tyAlmTxt := [(sAlmText:='Magazine Not Present'),(sAlmText:='Magazine 1 Is Empty'),(sAlmText:='Magazine 2 Is Empty'),(sAlmText:='Magazine 3 Is Empty'),(sAlmText:='Wrong Magazine Width On Position 4'),(sAlmText:='Wrong Magazine Height On Position 4'),(sAlmText:='Waiting for Unload Magazine 4'),2(0),91((0))];
END_VAR
(**)
(*Local Output*)
VAR
	sStepTxt : STRING[80];
	bPaused : BOOL;
END_VAR
(**)
VAR
	eBufferAct : eBufferAction;
	eSelClampCtrl : ePneuAction;
	eMagConv2ClpAct : eMagConv2ClpAction;
	eDSSMEMAAct : eSMEMAAction;
	eAGVMagAct : eAGVMagAction;
	eSafetyBarAct : ePneuAction;
	eUSSOTAct : eSOTAction;
	eDSSOTAct : eSOTAction;
END_VAR
(**)
VAR
	bOpsInitDone : BOOL;
	bMagBffrAvl : BOOL;
	bNewMagAllw : BOOL;
	bRlsMagAllw : BOOL;
	bStepMagExitedWait : BOOL;
	bStepMagVerification : BOOL;
	bStepMagMtyExit : BOOL;
	bStepMagUSCom : BOOL;
END_VAR
(**)
(*Local Input*)
VAR
	udiRstErr : UDINT := 0;
	bEn : BOOL := TRUE;
	bDis : BOOL := FALSE;
	bRun : BOOL;
	bStop : BOOL;
	bStep : BOOL;
	usiMagConv : USINT;
	bInfoEn : BOOL;
	bInfoMag1Mty : BOOL;
	bInfoMag2Mty : BOOL;
	bInfoMag3Mty : BOOL;
	a_bMagDis : ARRAY[1..4] OF BOOL;
	bNewMag : BOOL;
	bRlsMag : BOOL;
	tyBufferStat1 : tyBffrStat;
	tyBufferStat2 : tyBffrStat;
	tyBufferStat3 : tyBffrStat;
	tyBufferStat4 : tyBffrStat;
	bMagClampRS1 : BOOL;
	bMagClampRS2 : BOOL;
	bMagClampRS3 : BOOL;
	bMagClampRS4 : BOOL;
	bMagEntrySen1 : BOOL;
	bMagEntrySen2 : BOOL;
	bMagEntrySen3 : BOOL;
	bMagEntrySen4 : BOOL;
	bMagPresentSen1 : BOOL;
	bMagPresentSen2 : BOOL;
	bMagPresentSen3 : BOOL;
	bMagPresentSen4 : BOOL;
	bBufferMagPresent1 : BOOL;
	bBufferMagPresent2 : BOOL;
	bBufferMagPresent3 : BOOL;
	bBufferMagPresent4 : BOOL;
	dtBufferMagPresentTm1 : DATE_AND_TIME;
	dtBufferMagPresentTm2 : DATE_AND_TIME;
	dtBufferMagPresentTm3 : DATE_AND_TIME;
	dtBufferMagPresentTm4 : DATE_AND_TIME;
	eBufferStat : eBufferAction;
	eBufferStatus : eFBStatus;
	eMagConv2ClpStat : eMagConv2ClpAction;
	eMagConv2ClpStatus : eFBStatus;
	bMagConv2ClpHvMag : BOOL;
	eDSSMEMAStat : eSMEMAAction;
	eDSSMEMAStatus : eFBStatus;
	bDSSMEMAConvStart : BOOL;
	eAGVMagStat : eAGVMagAction;
	eAGVMagStatus : eFBStatus;
	bAGVMagMcRunRdy : BOOL;
	tyAGVToDTMag : tyTagAGVToDTMag;
	sProgNm : STRING[15] := 'Ops MagConvUL';
	bNtSettingsLoadDone : BOOL := TRUE;
END_VAR
(**)
(*Local*)
VAR
	bRstErr : BOOL;
	udiRstErrOld : UDINT;
	bInitDone : BOOL;
	bInitialDone : BOOL;
	eOpsStep : eMagConvLDStep := MagConvLDStepNA;
	eGotoOpsStep : eMagConvLDStep := MagSetupULStepInitPneu;
	bMagMtyExitedWait : BOOL;
	udi : UDINT;
	udi1 : UDINT;
	udiCount : UDINT;
	udiCmpTm : UDINT;
	udiMagAllwGo : UDINT;
	a_tyMagAllwBffrStat : ARRAY[1..4] OF tyBffrStat;
	a_bMagAllwMagClamped : ARRAY[1..4] OF BOOL;
	a_bMagAllwMagPresent : ARRAY[1..4] OF BOOL;
	a_udiMagAllwMagPresentTm : ARRAY[1..4] OF UDINT;
	a_udiMagAllwPriority : ARRAY[1..4] OF UDINT;
	a_udiMagAllwSum : ARRAY[1..4] OF UDINT;
	p_tyLocalBufferStat : REFERENCE TO tyBffrStat;
	p_bLocalMagEntrySen : REFERENCE TO BOOL;
	p_bLocalBufferMagPresent : REFERENCE TO BOOL;
	p_dtLocalBufferMagPresentTm : REFERENCE TO DATE_AND_TIME;
END_VAR
(**)
VAR
	fbWrongMagTm : TON := (PT:=T#5000ms);
	fbMagAutoDetTm : TON := (PT:=T#2000ms);
	fbMagRemovedTm : TON := (PT:=T#2000ms);
	fbEntSenOff : TON := (PT:=T#1000ms);
	fbVerifyWarningDelay : TON := (PT:=T#1000ms);
	bNewMagAutoDetected : BOOL;
	bNewMagVerified : BOOL;
	bNewMagVerifyStarted : BOOL;
	bIncorrectMagazineModel : BOOL;
	bSetMagFull : BOOL;
	bMagToAGVAvailable : BOOL;
	bWrongHeight : BOOL;
	bWrongWidth : BOOL;
	bMagSizeLarge : BOOL;
	bLimitSenActivated : BOOL;
END_VAR
VAR RETAIN
	bManualUnloadMag : BOOL;
END_VAR
VAR
	bAIVInPos : BOOL;
END_VAR
VAR RETAIN
	bMagExitedWait : BOOL;
END_VAR
VAR
	usiMagModel : USINT;
	bMagManEx : BOOL;
	bMagAutoEx : BOOL;
	bStepDSCom : BOOL;
	bOpsTravLifULUpdatePullSlot : BOOL;
	udiModuleNum : {REDUND_UNREPLICABLE} UDINT := 6071;
END_VAR
(**)
(**)
```

#### Act_Alarm.st
```iecst
(** 2019-03-25 **)
ACTION Act_Alarm:

	//Error
	IF EDGEPOS(eStatus = Error) THEN

		tyAlmData.sProgNm		:= p_sProgNm;
		tyAlmData.udiCode		:= udiStatus;
		tyAlmData.eSeverity		:= AlmSeverityError;
		tyAlmData.udiRunTime	:= tyAlmData.udiRunTime + 1;
		tyAlmData.bAlm			:= TRUE;
		tyAlmData.udiModuleNum  := udiModuleNum;
		g_sOpsMagConvLDProgNm	:= p_sProgNm;
		//Get Error Message
		IF tyAlmData.udiCode < 10000 OR tyAlmData.udiCode > 10099 THEN
			tyAlmData.sAlmMsg	:= 'Unknown';
			tyAlmData.sRcyMsg	:= 'Unknown';
		ELSE
			tyAlmData.sAlmMsg	:= a_tyAlmText[tyAlmData.udiCode].sAlmText;
			tyAlmData.sRcyMsg	:= a_tyAlmText[tyAlmData.udiCode].sRcyText;
		END_IF

	ELSIF bRstErr AND (tyAlmData.udiCode <> 0) THEN

		tyAlmData.udiCode		:= 0;
		tyAlmData.eSeverity		:= AlmSeverityNA;
		tyAlmData.sAlmMsg		:= '';
		tyAlmData.sRcyMsg		:= '';
		tyAlmData.bAlm			:= FALSE;
	END_IF

END_ACTION
```

#### Act_Background.st
```iecst
(** 2019-04-16 **)
ACTION Act_Background:

	//Reset bPaused
	IF EDGENEG(p_bStop OR p_bStep) THEN
		bPaused	:= FALSE;
	END_IF

	IF eStatus <> Error AND p_bRun = TRUE THEN
		IF (p_bEn = TRUE) AND (p_bDis = FALSE) THEN
			Act_OpsRun;
		ELSE
			bPaused	:= p_bStop OR p_bStep;
		END_IF

		IF EDGEPOS(p_bEn = FALSE OR p_bDis = TRUE) THEN
			Act_OpsRst;
		END_IF

	ELSIF eStatus <> Error THEN
		sStepTxt	:= 'Stop';
	ELSE
		sStepTxt	:= 'Error';
	END_IF

	//Reset
	IF EDGENEG(p_bRun) OR EDGEPOS(eStatus = Error) THEN
		Act_OpsInitial;
		Act_OpsRst;
	END_IF

	//Reset Error
	IF (eStatus = Error) AND bRstErr THEN
		eStatus		:= Idle;
		udiStatus	:= 0;
	END_IF

	//Always Run
//	IF NOT p_bRun AND bMagMtyExitedWait THEN
//		IF NOT p_bLocalMagEntrySen THEN
//			bMagMtyExitedWait	:= FALSE;
//		END_IF
//	END_IF

END_ACTION
```

#### Act_InitGlobal.st
```iecst
(** 2019-04-16 **)
ACTION Act_InitGlobal:

	(* Always Change If Project Change *)

	//Pass Data To Link
	p_bLinkDIMagPresentSen1 ACCESS p_DIMagPresentSen1;
	p_bLinkMagConv2Clp1MtrIn ACCESS p_MagConv2Clp1MtrSigOnOrLToR;
	p_bLinkMagConv2Clp1MtrOut ACCESS p_MagConv2Clp1MtrDirOrRToL;
	p_bLinkDIMagPresentSen2 ACCESS p_DIMagPresentSen2;
	p_bLinkMagConv2Clp2MtrIn ACCESS p_MagConv2Clp2MtrSigOnOrLToR;
	p_bLinkMagConv2Clp2MtrOut ACCESS p_MagConv2Clp2MtrDirOrRToL;
	p_bLinkDIMagPresentSen3 ACCESS p_DIMagPresentSen3;
	p_bLinkMagConv2Clp3MtrIn ACCESS p_MagConv2Clp3MtrSigOnOrLToR;
	p_bLinkMagConv2Clp3MtrOut ACCESS p_MagConv2Clp3MtrDirOrRToL;
	p_bLinkDIMagPresentSen3 ACCESS p_DIMagPresentSen3;
	p_bLinkMagConv2Clp3MtrIn ACCESS p_MagConv2Clp3MtrSigOnOrLToR;
	p_bLinkMagConv2Clp3MtrOut ACCESS p_MagConv2Clp3MtrDirOrRToL;
	p_bLinkDIMagPresentSen4 ACCESS p_DIMagPresentSen4;
	p_bLinkMagConv2Clp4MtrIn ACCESS p_MagConv2Clp4MtrSigOnOrLToR;
	p_bLinkMagConv2Clp4MtrOut ACCESS p_MagConv2Clp4MtrDirOrRToL;

	p_bLinkFixedMagClampRS1 ACCESS p_DIMag1FixedClampRS;
	p_bLinkRmtMagClampRS1 ACCESS p_DIMag1RemoteClampRS;

	p_bLinkFixedMagClampRS2 ACCESS p_DIMag2FixedClampRS;
	p_bLinkRmtMagClampRS2 ACCESS p_DIMag2RemoteClampRS;

	p_bLinkFixedMagClampRS3 ACCESS p_DIMag3FixedClampRS;
	p_bLinkRmtMagClampRS3 ACCESS p_DIMag3RemoteClampRS;

	p_bLinkFixedMagClampRS4 ACCESS p_DIMag4FixedClampRS;
	p_bLinkRmtMagClampRS4 ACCESS p_DIMag4RemoteClampRS;

	p_bLinkDIMagEntrySen ACCESS p_DIMagConvEntSen4;
	p_bLinkMcParamMagAutoDetTm ACCESS p_McParamMagAutoDetTm;
	p_bLinkNtParamMagModelAutoVerify ACCESS p_NtParamProjMagAutoVerifyPrep;
	p_bLinkMagRcpCurrRcpMagModel ACCESS p_MagRcpCurrRcpMagModel;

	p_bLinkNewMagVerified1 ACCESS p_OpsMagConvLD1NewMagVerified;
	p_bLinkNewMagVerified2 ACCESS p_OpsMagConvLD2NewMagVerified;
	p_bLinkNewMagVerified3 ACCESS p_OpsMagConvLD3NewMagVerified;

	p_eLinkMag ACCESS p_NtParamProjMag;
	p_usiLinkMod ACCESS p_ProdRcpCurrRcp1McMod;
	p_bLinkMagRcpCurrRcpMagModel1 ACCESS p_MagRcpCurrRcpMagModel1;

	p_eLinkMcParamMagExMode ACCESS p_McParamMagExMode;

	//Pass Data To Internal Use
	p_udiRstErr ACCESS p_RstErrReset;
	p_bEn ACCESS p_NtParamProjMag4ConvPrep;
	p_bRun ACCESS p_OpsRun;
	p_bStop ACCESS p_OpsStop;
	p_bStep ACCESS p_OpsStep;

	p_sProgNm ACCESS p_NtParamOpsMagConvLD4ProgNm;
	p_bNtSettingsLoadDone ACCESS p_StartupNtSettingsLoadDone;

	pa_bMagDis ACCESS p_OpsTravLifLDMagDis;

	p_bNewMag ACCESS p_UINewMag4;
	p_bRlsMag ACCESS p_UIRlsMag4;

	p_tyBufferStat1 ACCESS p_Buffer1BffrStat;
	p_tyBufferStat2 ACCESS p_Buffer2BffrStat;
	p_tyBufferStat3 ACCESS p_Buffer3BffrStat;
	p_tyBufferStat4 ACCESS p_Buffer4BffrStat;

	p_bMagEntrySen1 ACCESS p_DIMagConvEntSen1;
	p_bMagEntrySen2 ACCESS p_DIMagConvEntSen2;
	p_bMagEntrySen3 ACCESS p_DIMagConvEntSen3;
	p_bMagEntrySen4 ACCESS p_DIMagConvEntSen4;

	p_bMagPresentSen ACCESS p_Buffer4MagPresent;
	p_bBufferMagPresent1 ACCESS p_Buffer1MagPresent;
	p_bBufferMagPresent2 ACCESS p_Buffer2MagPresent;
	p_bBufferMagPresent3 ACCESS p_Buffer3MagPresent;
	p_bBufferMagPresent4 ACCESS p_Buffer4MagPresent;

	p_dtBufferMagPresentTm1 ACCESS p_Buffer1MagPresentTm;
	p_dtBufferMagPresentTm2 ACCESS p_Buffer2MagPresentTm;
	p_dtBufferMagPresentTm3 ACCESS p_Buffer3MagPresentTm;
	p_dtBufferMagPresentTm4 ACCESS p_Buffer4MagPresentTm;

	p_eBufferStat ACCESS p_Buffer4Stat;
	p_eBufferStatus ACCESS p_Buffer4Status;

	p_bBufferMagRemoved ACCESS p_Buffer4MagRemoved;

	p_eMagConv2ClpStat ACCESS p_MagConv2Clp4Stat;
	p_eMagConv2ClpStatus ACCESS p_MagConv2Clp4Status;
	p_bMagConv2ClpHvMag ACCESS p_MagConv2Clp4HvMag;

	p_eDSSMEMAStat ACCESS p_DSSMEMA4Stat;
	p_eDSSMEMAStatus ACCESS p_DSSMEMA4Status;
	p_bDSSMEMAConvStart ACCESS p_DSSMEMA4ConvStart;

	p_eAGVMagStat ACCESS p_AGVMag4Stat;
	p_eAGVMagStatus ACCESS p_AGVMag4Status;
	p_bAGVMagMcRunRdy ACCESS p_AGVMag4McRunRdy;
	p_tyAGVToDTMag ACCESS p_AGVTagAGVToDTMag;

	p_eSelClampCtrlStat ACCESS p_PneuNoSenSelClamp4Stat;
	p_eSelClampCtrlStatus ACCESS p_PneuNoSenSelClamp4Status;

	p_bDIMagConvHeightSen ACCESS p_DIMagConvHeightSen4;
	p_bDIMagConvSelUnclampRS ACCESS p_DIMag4SelUnclampRS;
	p_bDIMagConvCAB717Sen ACCESS p_DIMagConvCAB717MagSen4;
	p_bDIMagConvSmallSen ACCESS p_DIMagConvSmallMagSen4;
	p_bDIMagConvLargeSen ACCESS p_DIMagConvLargeMagSen4;
	p_bDIInShutterClosedRS ACCESS p_DIInShutterCloseRS;

	p_bOpsTravLifLDInitDone ACCESS p_OpsTravLifLDInitDone;

	//USSOT
	p_eUSSOTStat ACCESS p_USSOT4Stat;
	p_eUSSOTStatus ACCESS p_USSOT4Status;
	p_bUSSOTTransporting ACCESS p_USSOT4Transporting;
	p_bUSSOTConvStart ACCESS p_USSOT4ConvStart;
	p_bUSSOTConvStop ACCESS p_USSOT4ConvStop;
	p_bUSSOTUSRdy ACCESS p_USSOT4USRdy;
	p_bUSSOTUSLargeMagRdy ACCESS p_USSOT4USLargeMagRdy;

	//DSSOT
	p_eDSSOTStat ACCESS p_DSSOT4Stat;
	p_eDSSOTStatus ACCESS p_DSSOT4Status;
	p_bDSSOTConvStart ACCESS p_DSSOT4ConvStart;
	p_bDSSOTConvStop ACCESS p_DSSOT4ConvStop;

	p_bDISOTRcv ACCESS p_DISOT4Receive;

	p_bInShutterExtended ACCESS p_Pneu2SenInShutterExtended;

	p_bUSAllow ACCESS p_Follower1USAllow;

	p_bLD1ExitedWait ACCESS p_OpsMagConvLD1ExitedWait;
	p_bLD2ExitedWait ACCESS p_OpsMagConvLD2ExitedWait;
	p_bLD3ExitedWait ACCESS p_OpsMagConvLD3ExitedWait;

	p_eSafetyBarStat ACCESS p_Pneu2SMag4SafetyBarStat;
	p_eSafetyBarStatus ACCESS p_Pneu2SMag4SafetyBarStatus;
	p_bSafetyBarExtended ACCESS p_Pneu2SMag4SafetyBarExtended;
	p_bSafetyBarRetracted ACCESS p_Pneu2SMag4SafetyBarRetracted;

	p_bOpsTravLifULUpdatePullSlot ACCESS p_OpsTravLifULUpdatePullSlot;

	p_bProjLifTravMnlLoad	ACCESS p_NtParamProjLifTravMnlLoad;
	(* Always Change If Project Change *)

END_ACTION
```

#### Act_Initial.st
```iecst
(** 2019-01-20 **)
ACTION Act_Initial:

	//Initial
	IF p_bLinkDIMagPresentSen4 THEN
		bSetMagFull := TRUE;
	END_IF

END_ACTION
```

#### Act_InitLocal.st
```iecst
(** 2019-04-16 **)
ACTION Act_InitLocal:

	//Input Reference Link To Local Variable
	p_udiRstErr ACCESS ADR(udiRstErr);
	p_bEn ACCESS ADR(bEn);
	p_bDis ACCESS ADR(bDis);
	p_bRun ACCESS ADR(bRun);
	p_bStop ACCESS ADR(bStop);
	p_bStep ACCESS ADR(bStep);

	p_sProgNm ACCESS ADR(sProgNm);
	p_bNtSettingsLoadDone ACCESS ADR(bNtSettingsLoadDone);

	p_usiMagConv ACCESS ADR(usiMagConv);
	p_bInfoEn ACCESS ADR(bInfoEn);
	p_bInfoMag1Mty ACCESS ADR(bInfoMag1Mty);
	p_bInfoMag2Mty ACCESS ADR(bInfoMag2Mty);
	p_bInfoMag3Mty ACCESS ADR(bInfoMag3Mty);

	pa_bMagDis ACCESS ADR(a_bMagDis);

	p_bNewMag ACCESS ADR(bNewMag);
	p_bRlsMag ACCESS ADR(bRlsMag);

	p_tyBufferStat1 ACCESS ADR(tyBufferStat1);
	p_tyBufferStat2 ACCESS ADR(tyBufferStat2);
	p_tyBufferStat3 ACCESS ADR(tyBufferStat3);
	p_tyBufferStat4 ACCESS ADR(tyBufferStat4);

	p_bMagClampRS1 ACCESS ADR(bMagClampRS1);
	p_bMagClampRS2 ACCESS ADR(bMagClampRS2);
	p_bMagClampRS3 ACCESS ADR(bMagClampRS3);
	p_bMagClampRS4 ACCESS ADR(bMagClampRS4);

	p_bMagEntrySen1 ACCESS ADR(bMagEntrySen1);
	p_bMagEntrySen2 ACCESS ADR(bMagEntrySen2);
	p_bMagEntrySen3 ACCESS ADR(bMagEntrySen3);
	p_bMagEntrySen4 ACCESS ADR(bMagEntrySen4);

	p_bMagPresentSen1 ACCESS ADR(bMagPresentSen1);
	p_bMagPresentSen2 ACCESS ADR(bMagPresentSen2);
	p_bMagPresentSen3 ACCESS ADR(bMagPresentSen3);
	p_bMagPresentSen4 ACCESS ADR(bMagPresentSen4);

	p_bBufferMagPresent1 ACCESS ADR(bBufferMagPresent1);
	p_bBufferMagPresent2 ACCESS ADR(bBufferMagPresent2);
	p_bBufferMagPresent3 ACCESS ADR(bBufferMagPresent3);
	p_bBufferMagPresent4 ACCESS ADR(bBufferMagPresent4);

	p_dtBufferMagPresentTm1 ACCESS ADR(dtBufferMagPresentTm1);
	p_dtBufferMagPresentTm2 ACCESS ADR(dtBufferMagPresentTm2);
	p_dtBufferMagPresentTm3 ACCESS ADR(dtBufferMagPresentTm3);
	p_dtBufferMagPresentTm4 ACCESS ADR(dtBufferMagPresentTm4);

	p_eBufferStat ACCESS ADR(eBufferStat);
	p_eBufferStatus ACCESS ADR(eBufferStatus);

	p_eMagConv2ClpStat ACCESS ADR(eMagConv2ClpStat);
	p_eMagConv2ClpStatus ACCESS ADR(eMagConv2ClpStatus);
	p_bMagConv2ClpHvMag ACCESS ADR(bMagConv2ClpHvMag);

	p_eDSSMEMAStat ACCESS ADR(eDSSMEMAStat);
	p_eDSSMEMAStatus ACCESS ADR(eDSSMEMAStatus);
	p_bDSSMEMAConvStart ACCESS ADR(bDSSMEMAConvStart);

	p_eAGVMagStat ACCESS ADR(eAGVMagStat);
	p_eAGVMagStatus ACCESS ADR(eAGVMagStatus);
	p_bAGVMagMcRunRdy ACCESS ADR(bAGVMagMcRunRdy);
	p_tyAGVToDTMag ACCESS ADR(tyAGVToDTMag);

END_ACTION
```

#### Act_Link.st
```iecst
(** 2018-12-11 **)
ACTION Act_Link:

	IF p_eLinkMag = LDMagQuadruple = FALSE THEN
			//Sensor
			p_bMagPresentSen1	:= p_bLinkDIMagPresentSen1 OR p_bLinkMagConv2Clp1MtrIn OR p_bLinkMagConv2Clp1MtrOut;
			p_bMagPresentSen2	:= p_bLinkDIMagPresentSen2 OR p_bLinkMagConv2Clp2MtrIn OR p_bLinkMagConv2Clp2MtrOut;
			p_bMagPresentSen3	:= p_bLinkDIMagPresentSen3 OR p_bLinkMagConv2Clp3MtrIn OR p_bLinkMagConv2Clp3MtrOut;
			p_bMagPresentSen4	:= p_bLinkDIMagPresentSen4 OR p_bLinkMagConv2Clp4MtrIn OR p_bLinkMagConv2Clp4MtrOut;
			//Clamp RS
			p_bMagClampRS1 		:= (p_bLinkFixedMagClampRS1 AND p_bLinkRmtMagClampRS1) OR p_bLinkNewMagVerified1;
			p_bMagClampRS2		:= (p_bLinkFixedMagClampRS2 AND p_bLinkRmtMagClampRS2) OR p_bLinkNewMagVerified2;
			p_bMagClampRS3		:= (p_bLinkFixedMagClampRS3 AND p_bLinkRmtMagClampRS3) OR p_bLinkNewMagVerified3;
			p_bMagClampRS4		:= (p_bLinkFixedMagClampRS4 AND p_bLinkRmtMagClampRS4) OR bNewMagVerified;

	ELSE
		IF p_eLinkMag = LDMagQuadruple THEN
			CASE p_usiLinkMod OF
				0,1:

					//Sensor
					p_bMagPresentSen1	:= p_bLinkDIMagPresentSen1 OR p_bLinkMagConv2Clp1MtrIn OR p_bLinkMagConv2Clp1MtrOut;
					p_bMagPresentSen2	:= p_bLinkDIMagPresentSen2 OR p_bLinkMagConv2Clp2MtrIn OR p_bLinkMagConv2Clp2MtrOut;
					p_bMagPresentSen3	:= p_bLinkDIMagPresentSen3 OR p_bLinkMagConv2Clp3MtrIn OR p_bLinkMagConv2Clp3MtrOut;
					p_bMagPresentSen4	:= p_bLinkDIMagPresentSen4 OR p_bLinkMagConv2Clp4MtrIn OR p_bLinkMagConv2Clp4MtrOut;
					//Clamp RS
					p_bMagClampRS1 		:= (p_bLinkFixedMagClampRS1 AND p_bLinkRmtMagClampRS1) OR p_bLinkNewMagVerified1;
					p_bMagClampRS2		:= (p_bLinkFixedMagClampRS2 AND p_bLinkRmtMagClampRS2) OR p_bLinkNewMagVerified2;
					p_bMagClampRS3		:= (p_bLinkFixedMagClampRS3 AND p_bLinkRmtMagClampRS3) OR p_bLinkNewMagVerified3;
					p_bMagClampRS4		:= (p_bLinkFixedMagClampRS4 AND p_bLinkRmtMagClampRS4) OR bNewMagVerified;

				2:
					//Sensor
					p_bMagPresentSen1	:= FALSE;
					p_bMagPresentSen2	:= FALSE;
					p_bMagPresentSen3	:= p_bLinkDIMagPresentSen3 OR p_bLinkMagConv2Clp3MtrIn OR p_bLinkMagConv2Clp3MtrOut;
					p_bMagPresentSen4	:= p_bLinkDIMagPresentSen4 OR p_bLinkMagConv2Clp4MtrIn OR p_bLinkMagConv2Clp4MtrOut;
					//Clamp RS
					p_bMagClampRS1 		:= FALSE;
					p_bMagClampRS2		:= FALSE;
					p_bMagClampRS3		:= (p_bLinkFixedMagClampRS3 AND p_bLinkRmtMagClampRS3) OR p_bLinkNewMagVerified3;
					p_bMagClampRS4		:= (p_bLinkFixedMagClampRS4 AND p_bLinkRmtMagClampRS4) OR bNewMagVerified;
				END_CASE
		END_IF
	END_IF

	//Mag Exchange Mode
	CASE p_eLinkMcParamMagExMode OF
		McSetMagXcAutoManMode:
			bMagManEx := TRUE;
			bMagAutoEx := TRUE;

		McSetMagXcAutoMode:
			bMagManEx := FALSE;
			bMagAutoEx := TRUE;

		McSetMagXcManMode:
			bMagManEx := TRUE;
			bMagAutoEx := FALSE;

	END_CASE

	//New magazine auto detection at inlet sensor
	fbMagAutoDetTm(IN := p_bLinkDIMagEntrySen  OR p_bLinkDIMagPresentSen4, PT := DINT_TO_TIME(p_bLinkMcParamMagAutoDetTm));
	IF fbMagAutoDetTm.Q AND bMagManEx THEN
		bNewMagAutoDetected := TRUE;
	ELSE
		bNewMagAutoDetected := FALSE;
	END_IF

	//Front or rear lane magazine mode
	IF p_eLinkMag = LDMagQuadruple THEN
		CASE p_usiLinkMod OF
			0:
				usiMagModel := p_bLinkMagRcpCurrRcpMagModel;

			1,2:
				usiMagModel := p_bLinkMagRcpCurrRcpMagModel1;
		END_CASE

	ELSE
		usiMagModel := p_bLinkMagRcpCurrRcpMagModel;

	END_IF

	IF p_bLinkNtParamMagModelAutoVerify THEN
		IF usiMagModel = 0  //CAB706.2
			AND p_bDIMagConvHeightSen = TRUE
			AND p_bDIMagConvSelUnclampRS = FALSE
			AND p_bDIMagConvCAB717Sen = FALSE
			AND p_bDIMagConvSmallSen
			THEN
			bNewMagVerified:= TRUE;

		ELSIF  usiMagModel = 1 //CAB716.2
			AND p_bDIMagConvHeightSen = FALSE
			AND p_bDIMagConvSelUnclampRS = FALSE
			AND p_bDIMagConvCAB717Sen = FALSE
			AND p_bDIMagConvSmallSen
			THEN
			bNewMagVerified:= TRUE;

		ELSIF  usiMagModel = 2 //CAB717.2
			AND p_bDIMagConvHeightSen = FALSE
			AND p_bDIMagConvSelUnclampRS
			AND p_bDIMagConvCAB717Sen
			AND p_bDIMagConvLargeSen
			THEN
			bNewMagVerified:= TRUE;
		ELSE
			bNewMagVerified:= FALSE;
		END_IF
	ELSE
		bNewMagVerified:= TRUE;
	END_IF

	bAIVInPos := p_tyAGVToDTMag.bVEHInPos4 OR p_bDISOTRcv;

	IF p_bBufferMagRemoved THEN
		bManualUnloadMag := FALSE;
	END_IF

	IF EDGEPOS(p_bOpsTravLifULUpdatePullSlot) THEN
		bOpsTravLifULUpdatePullSlot := TRUE;
	ELSIF p_bOpsTravLifULUpdatePullSlot = FALSE THEN
		bOpsTravLifULUpdatePullSlot := FALSE;
	END_IF

END_ACTION
```

#### Init.st
```iecst
(** 2019-03-25 **)
PROGRAM _INIT

	(* Always Change If Project Change *)

	//Physical Configuration
	usiMagConv	:= 4;

	//Pass Address To Global Address For External Use
	//Action, State & Status

	//Alarm
	p_OpsMagConvLD4AlmData	:= ADR(tyAlmData);
	p_OpsMagConvLD4AlmData1	:= ADR(tyAlmData1);

	//Output
	p_OpsMagConvLD4StepTxt				:= ADR(sStepTxt);
	p_OpsMagConvLD4Paused				:= ADR(bPaused);

	p_OpsMagConvLD4BufferAct			:= ADR(eBufferAct);
	p_OpsMagConvLD4MagConv2ClpAct		:= ADR(eMagConv2ClpAct);
	p_OpsMagConvLD4DSSMEMAAct			:= ADR(eDSSMEMAAct);
	p_OpsMagConvLD4AGVMagAct			:= ADR(eAGVMagAct);
	p_OpsMagConvLD4SafetyBarAct			:= ADR(eSafetyBarAct);

	p_OpsMagConvLD4InitDone				:= ADR(bOpsInitDone);
	p_OpsMagConvLD4MagBffrAvl			:= ADR(bMagBffrAvl);
	p_OpsMagConvLD4NewMagAllw			:= ADR(bNewMagAllw);
	p_OpsMagConvLD4RlsMagAllw			:= ADR(bRlsMagAllw);
	p_OpsMagConvLD4StepMagExitedWait	:= ADR(bStepMagExitedWait);
	p_OpsMagConvLD4StepUSCom			:= ADR(bStepMagUSCom);

	p_OpsMagConvLD4StepSelClampCtrl		:= ADR(eSelClampCtrl);

	p_OpsMagConvLD4NewMagVerified		:= ADR(bNewMagVerified);
	p_OpsMagConvLD4MagMtyExit			:= ADR(bStepMagMtyExit);
	p_OpsMagConvLD4IncorrectMagModel    := ADR(bIncorrectMagazineModel);
	p_OpsMagConvLD4MagSizeL    			:= ADR(bMagSizeLarge);

	p_OpsMagConvLD4USSOTAct			:= ADR(eUSSOTAct);
	p_OpsMagConvLD4DSSOTAct			:= ADR(eDSSOTAct);

	p_OpsMagConvLD4ExitedWait			:= ADR(bMagExitedWait);
	p_OpsMagConvLD4DSCom				:= ADR(bStepDSCom);
	(* Always Change If Project Change *)

END_PROGRAM
```

#### Act_OpsInitial.st - Do Not Change!!!
```iecst
(** 2019-01-16 **)
ACTION Act_OpsInitial:

	eOpsStep		:= MagConvLDStepNA;
	eGotoOpsStep	:= MagConvLDStepInitMag;

	bOpsInitDone		:= FALSE;
	bMagBffrAvl			:= FALSE;
	bNewMagAllw			:= FALSE;
	bRlsMagAllw			:= FALSE;
	bStepMagExitedWait	:= FALSE;

END_ACTION
```

#### Act_OpsRun.st
```iecst
(** 2019-04-16 **)
ACTION Act_OpsRun:

	IF eGotoOpsStep <> eOpsStep THEN

		CASE eGotoOpsStep OF

			ELSE
				eOpsStep	:= eGotoOpsStep;

		END_CASE

	END_IF

	IF eOpsStep = eGotoOpsStep THEN

		IF bPaused = FALSE THEN

			CASE eOpsStep OF

				MagSetupULStepInitPneu:
					sStepTxt	:= 'Initializing Pneumatic';

					p_usiMagConv := 4;
					CASE p_usiMagConv OF
						1:
							p_tyLocalBufferStat ACCESS ADR(p_tyBufferStat1);
							p_bLocalMagEntrySen ACCESS ADR(p_bMagEntrySen1);
							p_bLocalBufferMagPresent ACCESS ADR(p_bBufferMagPresent1);
							p_dtLocalBufferMagPresentTm ACCESS ADR(p_dtBufferMagPresentTm1);
						2:
							p_tyLocalBufferStat ACCESS ADR(p_tyBufferStat2);
							p_bLocalMagEntrySen ACCESS ADR(p_bMagEntrySen2);
							p_bLocalBufferMagPresent ACCESS ADR(p_bBufferMagPresent2);
							p_dtLocalBufferMagPresentTm ACCESS ADR(p_dtBufferMagPresentTm2);
						3:
							p_tyLocalBufferStat ACCESS ADR(p_tyBufferStat4);
							p_bLocalMagEntrySen ACCESS ADR(p_bMagEntrySen3);
							p_bLocalBufferMagPresent ACCESS ADR(p_bBufferMagPresent3);
							p_dtLocalBufferMagPresentTm ACCESS ADR(p_dtBufferMagPresentTm3);
						4:
							p_tyLocalBufferStat ACCESS ADR(p_tyBufferStat4);
							p_bLocalMagEntrySen ACCESS ADR(p_bMagEntrySen4);
							p_bLocalBufferMagPresent ACCESS ADR(p_bBufferMagPresent4);
							p_dtLocalBufferMagPresentTm ACCESS ADR(p_dtBufferMagPresentTm4);
					END_CASE

					IF p_bProjLifTravMnlLoad = FALSE THEN
						eSafetyBarAct	:= PneuActExt;
					ELSE
						eGotoOpsStep := MagConvLDStepMagUSComm;
					END_IF

					IF (p_eSafetyBarStatus = Done AND p_eSafetyBarStat = PneuActExt) THEN
						eSafetyBarAct	:= PneuActIdle;
						eGotoOpsStep	:= MagConvLDStepInitMag;

						bPaused	:= p_bStop OR p_bStep;
					END_IF

				MagConvLDStepInitMag:
					sStepTxt	:= 'Initializing Magazine';

					IF p_bProjLifTravMnlLoad = TRUE THEN
						eGotoOpsStep := MagConvLDStepMagUSComm;
					ELSIF bMagExitedWait THEN
						eGotoOpsStep	:= MagConvLDStepInitMagEnt;
					ELSE
						//	eGotoOpsStep	:= MagConvLDStepInitMagConv;
						eGotoOpsStep	:= MagConvLDStepInitSetMagFull;
					END_IF

					bPaused	:= p_bStop OR p_bStep;

				MagConvLDStepInitMagEnt:
					sStepTxt	:= 'Initializing Magazine Conveyor';
					eMagConv2ClpAct	:= MagConv2ClpActInit;
					IF (p_eMagConv2ClpStatus = Done AND p_eMagConv2ClpStat = MagConv2ClpActInit) THEN
						eMagConv2ClpAct	:= MagConv2ClpActIdle;
						IF p_bMagConv2ClpHvMag = FALSE THEN
							eGotoOpsStep	:= MagConvLDStepMagUSComm;
						ELSE
							eGotoOpsStep	:= MagConvLDStepInitMagFixClp;
						END_IF
					END_IF

				MagConvLDStepInitMagFixClp:
					sStepTxt	:= 'Initializing Fixed Clamp';
					eMagConv2ClpAct	:= MagConv2ClpActFixClprClamp;
					IF (p_eMagConv2ClpStatus = Done AND p_eMagConv2ClpStat = MagConv2ClpActFixClprClamp) THEN
						eMagConv2ClpAct	:= MagConv2ClpActIdle;
						IF bMagAutoEx THEN
							eDSSOTAct	:= SOTActRun;
						ELSE
							eDSSOTAct	:= SOTActIdle;
						END_IF

						IF p_bDIMagConvCAB717Sen THEN
							bMagSizeLarge := TRUE;
						ELSE
							bMagSizeLarge := FALSE;
						END_IF
						eGotoOpsStep	:= MagConvLDStepSelClampCtrl;
					END_IF

				MagConvLDStepInitSetMagFull	:
					sStepTxt	:= 'Set Magazine Full';
					IF bSetMagFull AND p_tyBufferStat4.diTtlBrdCap = 1 THEN
						eBufferAct := BufferActSetFull;
					ELSIF p_eBufferStat = BufferActSetFull AND p_eBufferStatus = Done THEN
						bSetMagFull := FALSE;
						eBufferAct := BufferActIdle;
						eGotoOpsStep	:= MagConvLDStepInitMagConv;
					ELSIF bSetMagFull AND p_tyBufferStat4.diTtlBrdCap <> 1 THEN
						bSetMagFull := FALSE;
						eBufferAct := BufferActIdle;
						eGotoOpsStep	:= MagConvLDStepInitMagConv;
					ELSE
						bSetMagFull := FALSE;
						eBufferAct := BufferActIdle;
						eGotoOpsStep	:= MagConvLDStepInitMagConv;
					END_IF
					bPaused	:= p_bStop OR p_bStep;

				MagConvLDStepInitMagConv:
					sStepTxt	:= 'Initializing Magazine Conveyor';

					eMagConv2ClpAct	:= MagConv2ClpActInitStopClp;
					eSelClampCtrl := PneuActExt;

					IF (p_eMagConv2ClpStatus = Done AND p_eMagConv2ClpStat = MagConv2ClpActInitStopClp)
						AND (p_eSelClampCtrlStat = PneuActExt AND p_eSelClampCtrlStatus = Done)
						THEN
						eSelClampCtrl	:= PneuActIdle;
						eMagConv2ClpAct	:= MagConv2ClpActIdle;

						IF p_bMagConv2ClpHvMag = FALSE THEN
							eGotoOpsStep	:= MagConvLDStepMagUSComm;
						ELSE
						//	eGotoOpsStep		:= MagConvLDStepBffrStatChk;
							eGotoOpsStep		:= MagConvLDStepSelClampCtrl;
						END_IF

						bPaused	:= p_bStop OR p_bStep;

					END_IF

				MagConvLDStepSafetyBarExtCtrl:
					eSafetyBarAct	:= PneuActExt;

					IF(p_eSafetyBarStatus = Done AND p_eSafetyBarStat = PneuActExt)
						THEN
						eSafetyBarAct	:= PneuActIdle;
						eGotoOpsStep	:= MagConvLDStepMagUSComm;
					END_IF

				MagConvLDStepMagUSComm:
					sStepTxt	:= 'Communicating AIV And Ready Transport In Magazine';

					eAGVMagAct	:= AGVMagActEnter;
					IF bMagAutoEx THEN
						eUSSOTAct	:= SOTActRun;
					ELSE
						eUSSOTAct	:= SOTActIdle;
					END_IF
					eDSSOTAct	:= SOTActIdle;
					bMagSizeLarge := FALSE;
					bMagExitedWait	:= FALSE;

					IF p_bSafetyBarExtended = FALSE THEN
						eGotoOpsStep	:= MagConvLDStepSafetyBarExtCtrl;
					ELSIF p_bAGVMagMcRunRdy = TRUE OR p_bUSSOTTransporting= TRUE THEN
						eGotoOpsStep	:= MagConvLDStepMagEnt;

					ELSIF p_bNewMag = TRUE OR bNewMagAutoDetected = TRUE THEN
						eAGVMagAct		:= AGVMagActIdle;
						eGotoOpsStep	:= MagConvLDStepMagEntMnl;

					ELSE
						bPaused	:= p_bStop;

						IF bPaused = TRUE THEN
							eAGVMagAct	:= AGVMagActIdle;
							eUSSOTAct	:= SOTActIdle;
						END_IF

					END_IF

				MagConvLDStepMagEnt:

					IF p_bUSSOTConvStart THEN
						sStepTxt	:= 'Conveyor Entering Magazine To End';
						eMagConv2ClpAct	:= MagConv2ClpActEntStopClp;

					ELSIF bNewMagAutoDetected = TRUE THEN
						eAGVMagAct			:= AGVMagActIdle;
						eGotoOpsStep		:= MagConvLDStepMagEntMnl;

					ELSIF p_bUSSOTConvStop THEN
						sStepTxt	:= 'Conveyor Stopping';
						eMagConv2ClpAct	:= MagConv2ClpActStopClpr;
						IF (p_eMagConv2ClpStatus = Done AND p_eMagConv2ClpStat = MagConv2ClpActEntStopClp) THEN
							eMagConv2ClpAct		:= MagConv2ClpActIdle;

						END_IF
					END_IF

					IF (p_eMagConv2ClpStatus = Done AND p_eMagConv2ClpStat = MagConv2ClpActEntStopClp) THEN
						eAGVMagAct			:= AGVMagActIdle;
						eMagConv2ClpAct		:= MagConv2ClpActIdle;
						eUSSOTAct			:= SOTActIdle;
						eGotoOpsStep		:= MagConvLDStepSelClampCtrl;
						bPaused	:= p_bStop OR p_bStep;

					ELSE

					END_IF

				MagConvLDStepMagEntMnl:
					sStepTxt	:= 'Magazine Conveyor Entering Magazine Manually';
					IF p_bProjLifTravMnlLoad = FALSE THEN
						eMagConv2ClpAct		:= MagConv2ClpActEntStopClp;
					ELSE
						eGotoOpsStep		:= MagConvLDStepSelClampCtrl;
					END_IF
					IF p_eMagConv2ClpStatus = Done AND p_eMagConv2ClpStat = MagConv2ClpActEntStopClp THEN

						eMagConv2ClpAct		:= MagConv2ClpActIdle;
						eGotoOpsStep		:= MagConvLDStepSelClampCtrl;
						eUSSOTAct			:= SOTActIdle;
						eAGVMagAct			:= AGVMagActIdle;
						bPaused	:= p_bStop OR p_bStep;
					END_IF

				MagConvLDStepSelClampCtrl:
					sStepTxt	:= 'Magazine Selection Control';
					bNewMagVerifyStarted := TRUE;

					CASE p_bLinkMagRcpCurrRcpMagModel OF
						0: //CAB706.2
							IF p_bDIMagConvCAB717Sen = FALSE THEN
								eSelClampCtrl := PneuActRet;
							END_IF
							eGotoOpsStep	:= MagConvLDStepVerifyMag;

						1: //CAB716.2
							IF p_bDIMagConvCAB717Sen = FALSE THEN
								eSelClampCtrl := PneuActRet;
							END_IF
							eGotoOpsStep	:= MagConvLDStepVerifyMag;

						2: //CAB717.2
							eSelClampCtrl 	:= PneuActExt;
							eGotoOpsStep	:= MagConvLDStepVerifyMag;

					END_CASE

					bPaused	:= p_bStop OR p_bStep;

				MagConvLDStepVerifyMag:
					sStepTxt	:= 'Magazine Model Verification';

					bNewMagVerifyStarted := TRUE;
					fbWrongMagTm(IN:= bNewMagVerified = FALSE);
					IF fbWrongMagTm.Q AND NOT bMagExitedWait  THEN
						fbWrongMagTm(IN:= FALSE);
						eGotoOpsStep		:= MagConvLDStepMagExitMnl;
					ELSIF bMagExitedWait THEN
						eGotoOpsStep		:= MagConvLDStepMagExitMnl;
					ELSIF bNewMagVerified AND NOT bMagExitedWait THEN
						eSelClampCtrl	:= PneuActIdle;
						eGotoOpsStep		:= MagConvLDStepBffrStatChk;

					END_IF

					IF p_bDIMagConvCAB717Sen THEN
						bMagSizeLarge := TRUE;
					ELSE
						bMagSizeLarge := FALSE;
					END_IF

//					IF bNewMagVerified AND p_eSelClampCtrlStatus = Done THEN
//
//						eSelClampCtrl	:= PneuActIdle;
//						eGotoOpsStep	:= MagConvLDStepBffrStatChk;
//					END_IF
					bPaused	:= p_bStop OR p_bStep;

				MagConvLDStepBffrStatChk:
					sStepTxt	:= 'Checking Buffer Status';

					IF p_eBufferStatus = Idle THEN

						IF (p_tyLocalBufferStat.bBffrMty = TRUE OR p_bUSAllow = FALSE) THEN
							//eGotoOpsStep	:= MagConvLDStepMagMtyDSComm;
							eGotoOpsStep	:= MagConvLDStepMagExitClampCtrl;
						ELSE
							eGotoOpsStep	:= MagConvLDStepSafetyBarRetCtrl;
						END_IF

						bPaused	:= p_bStop OR p_bStep;

					END_IF

				MagConvLDStepSafetyBarRetCtrl:
					eSafetyBarAct	:= PneuActRet;

					IF (p_eSafetyBarStatus = Done AND p_eSafetyBarStat = PneuActRet) THEN
						eSafetyBarAct	:= PneuActIdle;
						eGotoOpsStep	:= MagConvLDStepPreNxtUnlBffr;

						bPaused	:= p_bStop OR p_bStep;
					END_IF

				MagConvLDStepPreNxtUnlBffr:
					sStepTxt	:= 'Computing Next Unload Buffer';

					eBufferAct	:= BufferActNxtUnload;

					IF p_eBufferStatus = Done AND p_eBufferStat = BufferActNxtUnload THEN
						eBufferAct		:= BufferActIdle;
						eGotoOpsStep	:= MagConvLDStepMagCmp;

						bPaused	:= p_bStop OR p_bStep;
					END_IF

				MagConvLDStepMagCmp:
					sStepTxt	:= 'Comparing Magazine';

					a_tyMagAllwBffrStat[1]	:= p_tyBufferStat1;
					a_tyMagAllwBffrStat[2]	:= p_tyBufferStat2;
					a_tyMagAllwBffrStat[3]	:= p_tyBufferStat3;
					a_tyMagAllwBffrStat[4]	:= p_tyBufferStat4;

					a_bMagAllwMagClamped[1]	:= p_bMagClampRS1;
					a_bMagAllwMagClamped[2]	:= p_bMagClampRS2;
					a_bMagAllwMagClamped[3]	:= p_bMagClampRS3;
					a_bMagAllwMagClamped[4]	:= p_bMagClampRS4;

					a_bMagAllwMagPresent[1]	:= p_bBufferMagPresent1 AND NOT p_bLD1ExitedWait;
					a_bMagAllwMagPresent[2]	:= p_bBufferMagPresent2 AND NOT p_bLD2ExitedWait;
					a_bMagAllwMagPresent[3]	:= p_bBufferMagPresent3 AND NOT p_bLD3ExitedWait;
					a_bMagAllwMagPresent[4]	:= p_bBufferMagPresent4 AND NOT bMagExitedWait;

					a_udiMagAllwMagPresentTm[1]	:= DT_TO_UDINT(p_dtBufferMagPresentTm1);
					a_udiMagAllwMagPresentTm[2]	:= DT_TO_UDINT(p_dtBufferMagPresentTm2);
					a_udiMagAllwMagPresentTm[3]	:= DT_TO_UDINT(p_dtBufferMagPresentTm3);
					a_udiMagAllwMagPresentTm[4]	:= DT_TO_UDINT(p_dtBufferMagPresentTm4);
					//Sorting Priority
					memset(ADR(a_udiMagAllwPriority), 0, SIZEOF(a_udiMagAllwPriority));

					FOR udi := 1 TO 4 DO
						udiCount	:= 4;
						udiCmpTm	:= a_udiMagAllwMagPresentTm[udi];

						FOR udi1 := 1 TO 4 DO
							IF a_udiMagAllwMagPresentTm[udi1] > udiCmpTm THEN
								udiCount	:= udiCount - 1;
							END_IF
						END_FOR

						a_udiMagAllwPriority[udi]	:= udiCount;
					END_FOR

					FOR udi := 4 TO 1 BY -1 DO
						FOR udi1 := 4 TO 1 BY -1 DO
							IF (udi <> udi1) AND (a_udiMagAllwPriority[udi] = a_udiMagAllwPriority[udi1]) THEN
								a_udiMagAllwPriority[udi1]	:= a_udiMagAllwPriority[udi1] - 1;
							END_IF
						END_FOR
					END_FOR

					//Checking Buffer Status
					memset(ADR(a_udiMagAllwSum), 0, SIZEOF(a_udiMagAllwSum));

					FOR udi := 1 TO 4 DO
						//Priority
						a_udiMagAllwSum[udi]	:= a_udiMagAllwSum[udi] + a_udiMagAllwPriority[udi];
						//Enable
						IF pa_bMagDis[udi] = FALSE THEN
							a_udiMagAllwSum[udi]	:= a_udiMagAllwSum[udi] + 1000;
						END_IF
						//Magazine Clamped
						IF a_bMagAllwMagClamped[udi] = TRUE THEN
							a_udiMagAllwSum[udi]	:= a_udiMagAllwSum[udi] + 1000;
						END_IF
						//Magazine Present
						IF a_bMagAllwMagPresent[udi] = TRUE THEN
							a_udiMagAllwSum[udi]	:= a_udiMagAllwSum[udi] + 1000;
						END_IF
						//Magazine Full
						IF a_tyMagAllwBffrStat[udi].bBffrFull = TRUE THEN
							a_udiMagAllwSum[udi]	:= a_udiMagAllwSum[udi] + 2500;
						END_IF
						//Magazine Available
						IF a_tyMagAllwBffrStat[udi].bBffrFull = FALSE AND a_tyMagAllwBffrStat[udi].bBffrMty = FALSE THEN
							a_udiMagAllwSum[udi]	:= a_udiMagAllwSum[udi] + 3000;
						END_IF

					END_FOR

					udiMagAllwGo	:= 99;

					FOR udi := 1 TO 4 DO
						//Enable + Magazine Clamped + Magazine Present + Magazine Available
						IF a_udiMagAllwSum[udi] >= 6000 THEN

							IF udiMagAllwGo <> 99 THEN
								//Priority
								IF a_udiMagAllwSum[udi] < a_udiMagAllwSum[udiMagAllwGo] THEN
									udiMagAllwGo	:= udi;
								END_IF
							ELSE
								udiMagAllwGo	:= udi;
							END_IF

						END_IF

					END_FOR

					IF udiMagAllwGo = 99 THEN

						FOR udi := 1 TO 4 DO
							//Enable + Magazine Clamped + Magazine Present + Magazine Full
							IF a_udiMagAllwSum[udi] >= 5500 THEN

								IF udiMagAllwGo <> 99 THEN
									//Priority
									IF a_udiMagAllwSum[udi] < a_udiMagAllwSum[udiMagAllwGo] THEN
										udiMagAllwGo	:= udi;
									END_IF
								ELSE
									udiMagAllwGo	:= udi;
								END_IF

							END_IF

						END_FOR

					END_IF

					IF p_bRlsMag = TRUE THEN
						eGotoOpsStep	:= MagConvLDStepMagExitMnl;

					ELSIF (p_tyLocalBufferStat.bBffrMty = TRUE OR p_bUSAllow = FALSE) AND p_bInShutterExtended THEN
					//	eGotoOpsStep    := MagConvLDStepMagMtyDSComm;
						eGotoOpsStep    := MagConvLDStepMagExitClampCtrl;
					ELSE

						IF udiMagAllwGo <> 99 THEN

							IF udiMagAllwGo = p_usiMagConv THEN
								bMagBffrAvl		:= TRUE;
								eGotoOpsStep	:= MagConvLDStepNxtUnloadBffr;

								bPaused	:= p_bStop OR p_bStep;
							ELSE
								bPaused	:= p_bStop;
							END_IF

						ELSE
							bPaused	:= p_bStop;
						END_IF

					END_IF

				MagConvLDStepNxtUnloadBffr:
					sStepTxt	:= 'Computing Next Unload Buffer';

					eBufferAct	:= BufferActNxtUnload;

					IF p_eBufferStatus = Done AND p_eBufferStat = BufferActNxtUnload THEN
						eBufferAct		:= BufferActIdle;
						eGotoOpsStep	:= MagConvLDStepBffrDSComm;

						bPaused	:= p_bStop OR p_bStep;
					END_IF

				MagConvLDStepBffrDSComm:
					sStepTxt	:= 'Communicating Buffer Downstream';

//					IF (p_tyBufferStat2.bBffrFull OR p_bBufferMagPresent2 = FALSE)
//						AND (p_tyBufferStat3.bBffrFull OR p_bBufferMagPresent3 = FALSE)
//						THEN
//						eDSSMEMAAct	:= SMEMAActRun;
//					END_IF

					eDSSMEMAAct	:= SMEMAActRun;

					IF p_bDSSMEMAConvStart = TRUE THEN
						eGotoOpsStep	:= MagConvLDStepBffrExitBrd;

					ELSIF bOpsTravLifULUpdatePullSlot THEN
						bMagBffrAvl		:= FALSE;
						IF p_tyLocalBufferStat.bBffrMty = FALSE THEN
							eGotoOpsStep	:= MagConvLDStepUnloadBffr;
						ELSE
							eGotoOpsStep	:= MagConvLDStepBffrStatChk;
							bMagBffrAvl		:= FALSE;
						END_IF

					ELSIF p_bRlsMag = TRUE THEN
						bMagBffrAvl		:= FALSE;
						eDSSMEMAAct		:= SMEMAActIdle;
						eGotoOpsStep	:= MagConvLDStepMagExitMnl;

					ELSIF (p_tyLocalBufferStat.bBffrMty = TRUE OR p_bUSAllow = FALSE) AND p_bInShutterExtended THEN
						bMagBffrAvl		:= FALSE;
						eDSSMEMAAct		:= SMEMAActIdle;
					//	eGotoOpsStep    := MagConvLDStepMagMtyDSComm;
						eGotoOpsStep    := MagConvLDStepMagExitClampCtrl;
					ELSE

						IF pa_bMagDis[usiMagConv] = TRUE THEN		//Checking Magazine Enable
							bMagBffrAvl		:= FALSE;
					//		eGotoOpsStep	:= MagConvLDStepMagCmp;
							eGotoOpsStep	:= MagConvLDStepPreNxtUnlBffr;

							bPaused	:= p_bStop OR p_bStep;
						ELSE
							bPaused	:= p_bStop;
						END_IF

						IF bPaused = TRUE OR pa_bMagDis[usiMagConv] = TRUE THEN
							eDSSMEMAAct	:= SMEMAActIdle;
						END_IF

					END_IF

				MagConvLDStepBffrExitBrd:
					IF p_bDSSMEMAConvStart = TRUE THEN
						sStepTxt	:= 'Transferring Board Out From Magazine';
						IF p_bRlsMag = TRUE THEN
							bMagBffrAvl		:= FALSE;
							eDSSMEMAAct		:= SMEMAActIdle;
							eGotoOpsStep	:= MagConvLDStepMagExitMnl;
						END_IF
					END_IF

					IF p_eDSSMEMAStatus = Done AND p_eDSSMEMAStat = SMEMAActRun THEN
						eDSSMEMAAct		:= SMEMAActIdle;
						//	eGotoOpsStep	:= MagConvLDStepUnloadBffr;
						IF p_tyLocalBufferStat.bBffrMty = FALSE THEN
							eGotoOpsStep	:= MagConvLDStepUnloadBffr;
						ELSE
							eGotoOpsStep	:= MagConvLDStepBffrStatChk;
							bMagBffrAvl		:= FALSE;
						END_IF
					END_IF

				MagConvLDStepUnloadBffr:
					sStepTxt	:= 'Unloading Buffer';

						eBufferAct	:= BufferActUnload;
						bOpsTravLifULUpdatePullSlot := FALSE;
						bMagBffrAvl		:= FALSE;
					IF p_eBufferStatus = Done AND p_eBufferStat = BufferActUnload THEN
						eBufferAct		:= BufferActIdle;
						bMagBffrAvl		:= FALSE;

							eGotoOpsStep	:= MagConvLDStepBffrStatChk;

						bPaused	:= p_bStop OR p_bStep;
					END_IF

				MagConvLDStepMagExitClampCtrl:
					sStepTxt	:= 'Extending Selection Clamp';
					eSelClampCtrl := PneuActExt;
					eSafetyBarAct	:= PneuActExt;

					IF (p_eSelClampCtrlStat = PneuActExt AND p_eSelClampCtrlStatus = Done)
						AND(p_eSafetyBarStatus = Done AND p_eSafetyBarStat = PneuActExt)
						THEN
							eSelClampCtrl	:= PneuActIdle;
							eSafetyBarAct	:= PneuActIdle;
							eGotoOpsStep    := MagConvLDStepMagMtyDSComm;
							bPaused	:= p_bStop OR p_bStep;
					END_IF

				MagConvLDStepMagMtyDSComm:
					sStepTxt	:= 'Communicating AGV Machine And Ready Exit';

					eAGVMagAct	:= AGVMagActExit;
					IF bMagAutoEx THEN
						eDSSOTAct	:= SOTActRun;
					ELSE
						eDSSOTAct	:= SOTActIdle;
					END_IF

					IF p_bAGVMagMcRunRdy = TRUE THEN
						eGotoOpsStep	:= MagConvLDStepMagMtyExit;

					ELSIF p_bRlsMag = TRUE OR ((p_tyLocalBufferStat.bBffrMty OR p_bUSAllow = FALSE) AND p_bInShutterExtended) THEN
						eAGVMagAct		:= AGVMagActIdle;
						eGotoOpsStep	:= MagConvLDStepMagExitMnl;

					ELSE
						bPaused	:= p_bStop;

						IF bPaused = TRUE THEN
							eAGVMagAct	:= AGVMagActIdle;
							eDSSOTAct	:= SOTActIdle;
						END_IF

					END_IF

				MagConvLDStepMagMtyExit:
					sStepTxt	:= 'Magazine Conveyor Exiting Magazine';

					eMagConv2ClpAct	:= MagConv2ClpActExitClpr;
					eSelClampCtrl	:= PneuActExt;

					IF ((p_eAGVMagStatus = Done AND p_eAGVMagStat = AGVMagActExit)
						OR (p_eDSSOTStatus = Done AND p_eDSSOTStat = SOTActRun))
						AND (p_eMagConv2ClpStatus = Done AND p_eMagConv2ClpStat = MagConv2ClpActExitClpr)
						AND (p_eSelClampCtrlStatus = Done AND p_eSelClampCtrlStat = PneuActExt)
						THEN

						eDSSOTAct	:= SOTActIdle;
						eAGVMagAct		:= AGVMagActIdle;
						eMagConv2ClpAct	:= MagConv2ClpActIdle;
						eSelClampCtrl	:= PneuActIdle;
						eGotoOpsStep	:= MagConvLDStepMagExitedAGVWait;
						bMagSizeLarge	:= FALSE;

						bPaused	:= p_bStop OR p_bStep;
					END_IF

				MagConvLDStepMagExitedAGVWait:
					sStepTxt	:= 'Magazine Exited and Wait for AGV Leave';

					IF bAIVInPos = FALSE OR p_bBufferMagRemoved THEN
						eGotoOpsStep	:= MagConvLDStepMagUSComm;
						eDSSOTAct	:= SOTActIdle;
					END_IF

					bPaused	:= p_bStop OR p_bStep;

				MagConvLDStepMagExitMnl:
					sStepTxt	:= 'Magazine Conveyor Exiting Magazine Manually';
					IF p_bProjLifTravMnlLoad = FALSE THEN
						eMagConv2ClpAct	:= MagConv2ClpActPreExitClpr;
						eSelClampCtrl	:= PneuActExt;
						eSafetyBarAct	:= PneuActExt;
					ELSE
						eGotoOpsStep    := MagConvLDStepMagExitedWait;
					END_IF
					IF (p_eMagConv2ClpStatus = Done AND p_eMagConv2ClpStat = MagConv2ClpActPreExitClpr)
						AND (p_eSelClampCtrlStatus = Done AND p_eSelClampCtrlStat = PneuActExt)
						AND (p_eSafetyBarStatus = Done AND p_eSafetyBarStat = PneuActExt)
						THEN
						eSelClampCtrl	:= PneuActIdle;
						eSafetyBarAct	:= PneuActIdle;
						eMagConv2ClpAct	:= MagConv2ClpActIdle;

						eGotoOpsStep	:= MagConvLDStepMagExitedWait;

						bPaused	:= p_bStop OR p_bStep;
					END_IF

				MagConvLDStepMagExitedWait:
					sStepTxt	:= 'Magazine Exited And Waiting For Remove';
					eAGVMagAct	:= AGVMagActExit;
					IF bMagAutoEx THEN
						eDSSOTAct	:= SOTActRun;
					ELSE
						eDSSOTAct	:= SOTActIdle;
					END_IF
					bMagExitedWait	:= TRUE;
					fbEntSenOff(IN:= p_bLocalMagEntrySen = FALSE);

					IF fbMagRemovedTm.Q OR fbEntSenOff.Q THEN
						bMagExitedWait	:= FALSE;
						eGotoOpsStep	:= MagConvLDStepMagUSComm;
						eDSSOTAct	:= SOTActIdle;

					ELSIF p_bNewMag = TRUE THEN
						bMagExitedWait	:= FALSE;
						eAGVMagAct	:= AGVMagActIdle;
						eGotoOpsStep	:= MagConvLDStepMagEntMnl;
						eDSSOTAct	:= SOTActIdle;
					END_IF

					IF p_bAGVMagMcRunRdy = TRUE THEN
						eGotoOpsStep	:= MagConvLDStepMagMtyExit;
					ELSIF p_bDSSOTConvStart = TRUE THEN
						eGotoOpsStep	:= MagConvLDStepMagMtyExit;
					END_IF

					bPaused	:= p_bStop OR p_bStep;

			END_CASE

		END_IF

	END_IF

	bNewMagAllw	:= eOpsStep = MagConvLDStepMagUSComm;
	bRlsMagAllw	:= (eOpsStep = MagConvLDStepMagCmp
					OR eOpsStep = MagConvLDStepBffrDSComm
					OR eOpsStep = MagConvLDStepMagMtyDSComm
					OR eOpsStep = MagConvLDStepBffrExitBrd)
					AND p_bDIInShutterClosedRS;

	Act_OpsInfo;

	//Operation State
	bOpsInitDone		:= eOpsStep > MagConvLDStepInitMagConv;
	bStepMagExitedWait	:= eOpsStep = MagConvLDStepMagExitedWait;
	bStepMagVerification:= eOpsStep = MagConvLDStepVerifyMag;
	bStepMagMtyExit:= eOpsStep = MagConvLDStepMagMtyExit;
	bStepMagUSCom := eOpsStep = MagConvLDStepMagUSComm;
	bStepDSCom 		:= eOpsStep = MagConvLDStepBffrDSComm;

END_ACTION
```

#### Act_OpsInfo.st
```iecst
ACTION Act_OpsInfo:

	//Reset
	udiStatus1	:= 0;

	//Magazine Verification Warning
	fbMagRemovedTm(IN:= p_bMagPresentSen = FALSE AND p_bLocalMagEntrySen = FALSE AND p_bBufferMagRemoved);
	IF fbMagRemovedTm.Q OR bNewMagVerified THEN
		bNewMagVerifyStarted := FALSE;
	END_IF

	fbVerifyWarningDelay(IN:= bNewMagVerifyStarted AND bNewMagVerified = FALSE AND bStepMagVerification = FALSE);

	IF fbVerifyWarningDelay.Q AND p_tyBufferStat4.bBffrMty = FALSE THEN
		IF bManualUnloadMag = FALSE THEN
			CASE usiMagModel OF
				0: //CAB706.2
					IF bWrongHeight THEN
						udiStatus1	:= 10005;
					ELSIF p_bDIMagConvHeightSen = FALSE THEN
						bWrongHeight := TRUE;

					ELSIF bWrongWidth THEN
						udiStatus1	:= 10004;
					ELSIF p_bDIMagConvSelUnclampRS
						OR p_bDIMagConvCAB717Sen
						OR p_bDIMagConvSmallSen = FALSE
						THEN
						bWrongWidth := TRUE;
					END_IF

				1: //CAB716.2
					IF bWrongHeight THEN
						udiStatus1	:= 10005;
					ELSIF p_bDIMagConvHeightSen = TRUE THEN
						bWrongHeight := TRUE;

					ELSIF bWrongWidth THEN
						udiStatus1	:= 10004;
					ELSIF p_bDIMagConvSelUnclampRS
						OR p_bDIMagConvCAB717Sen
						OR p_bDIMagConvSmallSen = FALSE
						THEN
						bWrongWidth := TRUE;
					END_IF

				2: //CAB717.2
					IF bWrongHeight THEN
						udiStatus1	:= 10005;
					ELSIF p_bDIMagConvHeightSen THEN
						bWrongHeight := TRUE;

					ELSIF bWrongWidth THEN
						udiStatus1	:= 10004;
					ELSIF p_bDIMagConvSelUnclampRS = FALSE
						OR p_bDIMagConvCAB717Sen = FALSE
						OR p_bDIMagConvLargeSen
						THEN
						bWrongWidth := TRUE;

					END_IF

			END_CASE
		ELSIF bManualUnloadMag THEN
			udiStatus1	:= 10006;
		END_IF

	ELSIF 	udiStatus1 <> 10004
		AND udiStatus1 <> 10005
		AND p_tyBufferStat4.bBffrMty = FALSE
		AND bStepMagExitedWait
		AND p_bLocalMagEntrySen
		THEN
		udiStatus1	:= 10006;
		bManualUnloadMag := TRUE;
	ELSE
		bWrongHeight := FALSE;
		bWrongWidth	:= FALSE;
	END_IF

	bIncorrectMagazineModel := udiStatus1 = 10004 OR udiStatus1 = 10005;

END_ACTION
```

#### Act_OpsRst.st - Do Not Change!!!
```iecst
(** 2019-03-25 **)
ACTION Act_OpsRst:

	udiStatus1	:= 0;

	eBufferAct		:= BufferActIdle;
	eMagConv2ClpAct	:= MagConv2ClpActIdle;
	eDSSMEMAAct		:= SMEMAActIdle;
	eAGVMagAct		:= AGVMagActIdle;
	eSelClampCtrl	:= PneuActIdle;
	eDSSOTAct		:= SOTActIdle;
	eUSSOTAct		:= SOTActIdle;
	eSafetyBarAct	:= PneuActIdle;

	bNewMagVerified := FALSE;
	bNewMagVerifyStarted := FALSE;

END_ACTION
```

### OpsLifMagLD.typ - Do Not Change!!!
```iecst
(*2018-12-11*)
(**)
(*Sequence*)

TYPE
	eLifMagLDStep :
		(
		LifMagLDStepNA,
		LifMagLDStepInitLif,
		LifMagLDStepMagCmp,
		LifMagLDStepNxtUnloadBffr,
		LifMagLDStepLifMov,
		LifMagLDStepBffrDSComm,
		LifMagLDStepBffrExitBrd,
		LifMagLDStepUnloadBffr,
		LifMagLDStepLifMovUnloadMag,
		LifMagLDStepUnloadMag
		);
	eLifMagLDStep1 :
		(
		LifMagLDStep1NA,
		LifMagLDStep1InitLif,
		LifMagLDStep1MagCmp,
		LifMagLDStep1NxtUnloadBffr,
		LifMagLDStep1PreLifMov,
		LifMagLDStep1LifMov,
		LifMagLDStep1BffrDSComm,
		LifMagLDStep1BffrExitLifMovWait,
		LifMagLDStep1BffrExitLifMov,
		LifMagLDStep1BffrExitBrd,
		LifMagLDStep1UnloadBffr,
		LifMagLDStep1LifMovUnloadMag,
		LifMagLDStep1UnloadMag
		);
	eLifMagLDMagNxtUnload :
		(
		MagNxtUnloadInvalid,
		MagNxtUnloadMag1,
		MagNxtUnloadMag2,
		MagNxtUnloadMag3
		);
END_TYPE
```

### OpsLifMagLD.var - Change By Project
```iecst
(*2019-03-25*)
(**)
(*Action & State & Status*)
(**)
(*Alarm*)
VAR
	p_OpsLifMagLDAlmData : UDINT;
	p_OpsLifMagLDAlmData1 : UDINT;
END_VAR
(**)
(*Output*)
VAR
	p_OpsLifMagLDStepTxt : UDINT;
	p_OpsLifMagLDPaused : UDINT;
END_VAR
(**)
VAR
	p_OpsLifMagLDLifterAct : UDINT;
	p_OpsLifMagLDBufferAct1 : UDINT;
	p_OpsLifMagLDBufferAct2 : UDINT;
	p_OpsLifMagLDBufferAct3 : UDINT;
	p_OpsLifMagLDDSSMEMAAct1 : UDINT;
	p_OpsLifMagLDDSSMEMAAct2 : UDINT;
	p_OpsLifMagLDDSSMEMAAct3 : UDINT;
END_VAR
(**)
VAR
	p_OpsLifMagLDGoUnloadSlt1 : UDINT;
	p_OpsLifMagLDGoUnloadSlt2 : UDINT;
	p_OpsLifMagLDGoUnloadSlt3 : UDINT;
	p_OpsLifMagLDMagNxtUnload : UDINT;
	p_OpsLifMagLDBffrExitBrd : UDINT;
	p_OpsLifMagLDUnloadingMov : UDINT;
	p_OpsLifMagLDUnloading : UDINT;
END_VAR
```

### Program Logical/Operations/OpsLifMagLD (IEC) - 1.00.0 - 

#### InputRef.var
```iecst
(*2019-04-16*)
(**)
(*General*)
VAR
	p_udiRstErr : REFERENCE TO UDINT;
	p_bEn : REFERENCE TO BOOL;
	p_bDis : REFERENCE TO BOOL;
	p_bRun : REFERENCE TO BOOL;
	p_bStop : REFERENCE TO BOOL;
	p_bStep : REFERENCE TO BOOL;
END_VAR
(**)
(*Configuration*)
VAR
	p_sProgNm : REFERENCE TO STRING[15];
	p_bNtSettingsLoadDone : REFERENCE TO BOOL;
END_VAR
(**)
VAR
	pa_bMagDis : REFERENCE TO ARRAY[1..3] OF BOOL;
	p_bUnloadMag : REFERENCE TO BOOL;
	p_bDSAllow : REFERENCE TO BOOL;
	p_bPullerRotCylPrep : REFERENCE TO BOOL;
	p_bPullerNoRotCylExitStartLif : REFERENCE TO BOOL;
	p_diPullerExtMaxSlt : REFERENCE TO DINT;
	p_diPullerExtMinSlt : REFERENCE TO DINT;
	p_bLifterSafeInitialize : REFERENCE TO BOOL;
END_VAR
(**)
VAR
	p_bProdRcpCurrRcpTopToBtm : REFERENCE TO BOOL;
	p_diProdRcpCurrRcpPitch : REFERENCE TO DINT;
END_VAR
(**)
VAR
	p_bMagSetupDone1 : REFERENCE TO BOOL;
	p_bMagSetupDone2 : REFERENCE TO BOOL;
	p_bMagSetupDone3 : REFERENCE TO BOOL;
END_VAR
(**)
VAR
	p_tyBufferStat1 : REFERENCE TO tyBffrStat;
	p_tyBufferStat2 : REFERENCE TO tyBffrStat;
	p_tyBufferStat3 : REFERENCE TO tyBffrStat;
END_VAR
(**)
VAR
	p_bMagPresentSen1 : REFERENCE TO BOOL;
	p_bMagPresentSen2 : REFERENCE TO BOOL;
	p_bMagPresentSen3 : REFERENCE TO BOOL;
END_VAR
(**)
VAR
	p_bBufferMagPresent1 : REFERENCE TO BOOL;
	p_bBufferMagPresent2 : REFERENCE TO BOOL;
	p_bBufferMagPresent3 : REFERENCE TO BOOL;
END_VAR
(**)
VAR
	p_dtBufferMagPresentTm1 : REFERENCE TO DATE_AND_TIME;
	p_dtBufferMagPresentTm2 : REFERENCE TO DATE_AND_TIME;
	p_dtBufferMagPresentTm3 : REFERENCE TO DATE_AND_TIME;
END_VAR
(**)
VAR
	p_eLifterStat : REFERENCE TO eLifterAction;
	p_eLifterStatus : REFERENCE TO eFBStatus;
END_VAR
(**)
VAR
	p_eBufferStat1 : REFERENCE TO eBufferAction;
	p_eBufferStatus1 : REFERENCE TO eFBStatus;
END_VAR
(**)
VAR
	p_eBufferStat2 : REFERENCE TO eBufferAction;
	p_eBufferStatus2 : REFERENCE TO eFBStatus;
END_VAR
(**)
VAR
	p_eBufferStat3 : REFERENCE TO eBufferAction;
	p_eBufferStatus3 : REFERENCE TO eFBStatus;
END_VAR
(**)
VAR
	p_eDSSMEMAStat1 : REFERENCE TO eSMEMAAction;
	p_eDSSMEMAStatus1 : REFERENCE TO eFBStatus;
	p_bDSSMEMAConvStart1 : REFERENCE TO BOOL;
END_VAR
(**)
VAR
	p_eDSSMEMAStat2 : REFERENCE TO eSMEMAAction;
	p_eDSSMEMAStatus2 : REFERENCE TO eFBStatus;
	p_bDSSMEMAConvStart2 : REFERENCE TO BOOL;
END_VAR
(**)
VAR
	p_eDSSMEMAStat3 : REFERENCE TO eSMEMAAction;
	p_eDSSMEMAStatus3 : REFERENCE TO eFBStatus;
	p_bDSSMEMAConvStart3 : REFERENCE TO BOOL;
END_VAR
(**)
(*Magazine*)
VAR
	p_diBufferNxtUnloadSlt1 : REFERENCE TO DINT;
	p_diBufferNxtUnloadSlt2 : REFERENCE TO DINT;
	p_diBufferNxtUnloadSlt3 : REFERENCE TO DINT;
END_VAR
```

#### InputRef_Link.var
```iecst
(*2022-03-17*)
(**)
VAR
	p_bLinkPullerRetRS : REFERENCE TO BOOL;
	p_bLinkInShutterCloRS : REFERENCE TO BOOL;
	p_bLinkInShutterExtended : REFERENCE TO BOOL;
END_VAR
```

#### Local.var
```iecst
(*2019-04-16*)
(**)
(*Local Action, State & Status*)
VAR
	eStatus : eFBStatus := Idle;
	udiStatus : UDINT := 0;
	udiStatus1 : UDINT := 0;
END_VAR
(**)
(*Local Alarm*)
VAR
	tyAlmData : tyAlmDat;
	tyAlmData1 : tyAlmDat;
	a_tyAlmText : ARRAY[10000..10099] OF tyAlmTxt := [(sAlmText:='Magazine Not Present'),(sAlmText:='Magazine 1 Is Empty'),(sAlmText:='Magazine 2 Is Empty'),(sAlmText:='Magazine 3 Is Empty'),(sAlmText:='Lifter Pre-Exit Position Are Invalid',sRcyText:='Reset And Resume Operation. If The Problem Persists, Please Contact Nutek For A Possible Solution.'),(sAlmText:='Lifter Exit Position Are Invalid',sRcyText:='Reset And Resume Operation. If The Problem Persists, Please Contact Nutek For A Possible Solution.'),94(0)];
END_VAR
(**)
(*Local Output*)
VAR
	sStepTxt : STRING[80];
	bPaused : BOOL;
END_VAR
(**)
VAR
	eLifterAct : eLifterAction;
	eBufferAct1 : eBufferAction;
	eBufferAct2 : eBufferAction;
	eBufferAct3 : eBufferAction;
	eDSSMEMAAct1 : eSMEMAAction;
	eDSSMEMAAct2 : eSMEMAAction;
	eDSSMEMAAct3 : eSMEMAAction;
END_VAR
(**)
VAR
	diGoUnloadSlt1 : DINT;
	diGoUnloadSlt2 : DINT;
	diGoUnloadSlt3 : DINT;
	eMagNxtUnload : eLifMagLDMagNxtUnload;
	bBffrExitBrd : BOOL;
	bUnloadingMov : BOOL;
	bUnloading : BOOL;
END_VAR
(**)
(*Local Input*)
VAR
	udiRstErr : UDINT := 0;
	bEn : BOOL := TRUE;
	bDis : BOOL := TRUE;
	bRun : BOOL;
	bStop : BOOL;
	bStep : BOOL;
	a_bMagDis : ARRAY[1..3] OF BOOL;
	bUnloadMag : BOOL;
	bDSAllow : BOOL := TRUE;
	bPullerRotCylPrep : BOOL;
	bPullerNoRotCylExitStartLif : BOOL;
	diPullerExtMaxSlt : DINT;
	diPullerExtMinSlt : DINT;
	bLifterSafeInitialize : BOOL := TRUE;
	bProdRcpCurrRcpTopToBtm : BOOL;
	diProdRcpCurrRcpPitch : DINT;
	bMagSetupDone1 : BOOL := TRUE;
	bMagSetupDone2 : BOOL := TRUE;
	bMagSetupDone3 : BOOL := TRUE;
	tyBufferStat1 : tyBffrStat;
	tyBufferStat2 : tyBffrStat;
	tyBufferStat3 : tyBffrStat;
	bMagPresentSen1 : BOOL;
	bMagPresentSen2 : BOOL;
	bMagPresentSen3 : BOOL;
	bBufferMagPresent1 : BOOL;
	bBufferMagPresent2 : BOOL;
	bBufferMagPresent3 : BOOL;
	dtBufferMagPresentTm1 : DATE_AND_TIME;
	dtBufferMagPresentTm2 : DATE_AND_TIME;
	dtBufferMagPresentTm3 : DATE_AND_TIME;
	eLifterStat : eLifterAction;
	eLifterStatus : eFBStatus;
	eBufferStat1 : eBufferAction;
	eBufferStatus1 : eFBStatus;
	eBufferStat2 : eBufferAction;
	eBufferStatus2 : eFBStatus;
	eBufferStat3 : eBufferAction;
	eBufferStatus3 : eFBStatus;
	eDSSMEMAStat1 : eSMEMAAction;
	eDSSMEMAStatus1 : eFBStatus;
	bDSSMEMAConvStart1 : BOOL;
	eDSSMEMAStat2 : eSMEMAAction;
	eDSSMEMAStatus2 : eFBStatus;
	bDSSMEMAConvStart2 : BOOL;
	eDSSMEMAStat3 : eSMEMAAction;
	eDSSMEMAStatus3 : eFBStatus;
	bDSSMEMAConvStart3 : BOOL;
	diBufferNxtUnloadSlt1 : DINT;
	diBufferNxtUnloadSlt2 : DINT;
	diBufferNxtUnloadSlt3 : DINT;
	sProgNm : STRING[15] := 'Ops LifMagUL';
	bNtSettingsLoadDone : BOOL := TRUE;
END_VAR
(**)
(*Local*)
VAR
	bRstErr : BOOL;
	udiRstErrOld : UDINT;
	bInitDone : BOOL;
	bInitialDone : BOOL;
	eOpsStep : eLifMagLDStep := LifMagLDStepNA;
	eGotoOpsStep : eLifMagLDStep := LifMagLDStepInitLif;
	eOpsStep1 : eLifMagLDStep1 := LifMagLDStep1NA;
	eGotoOpsStep1 : eLifMagLDStep1 := LifMagLDStep1InitLif;
	udi : UDINT;
	udi1 : UDINT;
	udiCount : UDINT;
	udiCmpTm : UDINT;
	udiMagAllwGo : UDINT;
	a_bMagAllwMagSetupDone : ARRAY[1..3] OF BOOL;
	a_tyMagAllwBffrStat : ARRAY[1..3] OF tyBffrStat;
	a_bMagAllwMagPresent : ARRAY[1..3] OF BOOL;
	a_udiMagAllwMagPresentTm : ARRAY[1..3] OF UDINT;
	a_udiMagAllwPriority : ARRAY[1..3] OF UDINT;
	a_udiMagAllwSum : ARRAY[1..3] OF UDINT;
	udiModuleNum : {REDUND_UNREPLICABLE} UDINT := 6091;
	p_tyLocalBufferStat : REFERENCE TO tyBffrStat;
	p_bLocalBufferMagPresent : REFERENCE TO BOOL;
	p_dtLocalBufferMagPresentTm : REFERENCE TO DATE_AND_TIME;
	p_eLocalBufferAct : REFERENCE TO eBufferAction;
	p_eLocalBufferStat : REFERENCE TO eBufferAction;
	p_eLocalBufferStatus : REFERENCE TO eFBStatus;
	p_eLocalDSSMEMAAct : REFERENCE TO eSMEMAAction;
	p_eLocalDSSMEMAStat : REFERENCE TO eSMEMAAction;
	p_eLocalDSSMEMAStatus : REFERENCE TO eFBStatus;
	p_bLocalDSSMEMAConvStart : REFERENCE TO BOOL;
END_VAR
```

#### Act_Alarm.st
```iecst
(** 2019-03-25 **)
ACTION Act_Alarm:

	//Error
	IF EDGEPOS(eStatus = Error) THEN

		tyAlmData.sProgNm		:= p_sProgNm;
		tyAlmData.udiCode		:= udiStatus;
		tyAlmData.eSeverity		:= AlmSeverityError;
		tyAlmData.udiRunTime	:= tyAlmData.udiRunTime + 1;
		tyAlmData.bAlm			:= TRUE;
		tyAlmData.udiModuleNum  := udiModuleNum;
		g_sOpsLifMagLDProgNm	:= p_sProgNm;
		//Get Error Message
		IF tyAlmData.udiCode < 10000 OR tyAlmData.udiCode > 10099 THEN
			tyAlmData.sAlmMsg	:= 'Unknown';
			tyAlmData.sRcyMsg	:= 'Unknown';
		ELSE
			tyAlmData.sAlmMsg	:= a_tyAlmText[tyAlmData.udiCode].sAlmText;
			tyAlmData.sRcyMsg	:= a_tyAlmText[tyAlmData.udiCode].sRcyText;
		END_IF

	ELSIF bRstErr AND (tyAlmData.udiCode <> 0) THEN

		tyAlmData.udiCode		:= 0;
		tyAlmData.eSeverity		:= AlmSeverityNA;
		tyAlmData.sAlmMsg		:= '';
		tyAlmData.sRcyMsg		:= '';
		tyAlmData.bAlm			:= FALSE;
	END_IF

END_ACTION
```

#### Act_InitGlobal.st
```iecst
(** 2019-04-16 **)
ACTION Act_InitGlobal:

	(* Always Change If Project Change *)

	//Pass Data To Link
	p_bLinkPullerRetRS ACCESS p_DIPullerRetRS; //safeinitial param
	p_bLinkInShutterCloRS ACCESS p_DIInShutterCloseRS; //safeinitial param
	p_bLinkInShutterExtended ACCESS p_Pneu2SenInShutterExtended;

	//Pass Data To Internal Use
	p_udiRstErr ACCESS p_RstErrReset;
	p_bRun ACCESS p_OpsRun;
	p_bStop ACCESS p_OpsStop;
	p_bStep ACCESS p_OpsStep;

	p_sProgNm ACCESS p_NtParamOpsLifMagLDProgNm;
	p_bNtSettingsLoadDone ACCESS p_StartupNtSettingsLoadDone;

	pa_bMagDis ACCESS p_OpsTravLifLDMagDis;
	p_bUnloadMag ACCESS p_UIUnloadMag;
	p_bPullerRotCylPrep ACCESS p_NtParamProjPullerRotCylPrep;
	p_bPullerNoRotCylExitStartLif ACCESS p_Pneu2SenPullerExtended;
	p_diPullerExtMaxSlt ACCESS p_NtParamProjPullerExtMaxSlt;
	p_diPullerExtMinSlt ACCESS p_NtParamProjPullerExtMinSlt;

	p_bProdRcpCurrRcpTopToBtm ACCESS p_ProdRcpCurrRcp1TopToBtm;
	p_diProdRcpCurrRcpPitch ACCESS p_ProdRcpCurrRcp1Pitch;

	p_tyBufferStat1 ACCESS p_Buffer1BffrStat;
	p_tyBufferStat2 ACCESS p_Buffer2BffrStat;
	p_tyBufferStat3 ACCESS p_Buffer3BffrStat;

	p_bMagPresentSen1 ACCESS p_DIMagPresentSen1;
	p_bMagPresentSen2 ACCESS p_DIMagPresentSen2;
	p_bMagPresentSen3 ACCESS p_DIMagPresentSen3;

	p_bBufferMagPresent1 ACCESS p_Buffer1MagPresent;
	p_bBufferMagPresent2 ACCESS p_Buffer2MagPresent;
	p_bBufferMagPresent3 ACCESS p_Buffer3MagPresent;

	p_dtBufferMagPresentTm1 ACCESS p_Buffer1MagPresentTm;
	p_dtBufferMagPresentTm2 ACCESS p_Buffer2MagPresentTm;
	p_dtBufferMagPresentTm3 ACCESS p_Buffer3MagPresentTm;

	p_eLifterStat ACCESS p_LifterBtmStat;
	p_eLifterStatus ACCESS p_LifterBtmStatus;

	p_eBufferStat1 ACCESS p_Buffer1Stat;
	p_eBufferStatus1 ACCESS p_Buffer1Status;

	p_eBufferStat2 ACCESS p_Buffer2Stat;
	p_eBufferStatus2 ACCESS p_Buffer2Status;

	p_eBufferStat3 ACCESS p_Buffer3Stat;
	p_eBufferStatus3 ACCESS p_Buffer3Status;

	p_eDSSMEMAStat1 ACCESS p_DSSMEMA1Stat;
	p_eDSSMEMAStatus1 ACCESS p_DSSMEMA1Status;
	p_bDSSMEMAConvStart1 ACCESS p_DSSMEMA1ConvStart;

	p_eDSSMEMAStat2 ACCESS p_DSSMEMA2Stat;
	p_eDSSMEMAStatus2 ACCESS p_DSSMEMA2Status;
	p_bDSSMEMAConvStart2 ACCESS p_DSSMEMA2ConvStart;

	p_eDSSMEMAStat3 ACCESS p_DSSMEMA3Stat;
	p_eDSSMEMAStatus3 ACCESS p_DSSMEMA3Status;
	p_bDSSMEMAConvStart3 ACCESS p_DSSMEMA3ConvStart;

	p_diBufferNxtUnloadSlt1 ACCESS p_Buffer1NxtUnloadSlt;
	p_diBufferNxtUnloadSlt2 ACCESS p_Buffer2NxtUnloadSlt;
	p_diBufferNxtUnloadSlt3 ACCESS p_Buffer3NxtUnloadSlt;

	(* Always Change If Project Change *)

END_ACTION
```
